LIN {X 0,Y 573.263,Z 117.071,A -85,B 0,C 180,E1 -2310.634,E2 -2310.634} C_VEL
LIN {X 0,Y 573.25,Z 117.074,A -85,B 0,C 180,E1 -2313.024,E2 -2313.024} C_VEL
LIN {X 0,Y 573.273,Z 117.075,A -85,B 0,C 180,E1 -2315.366,E2 -2315.366} C_VEL
LIN {X 0,Y 573.228,Z 117.075,A -85,B 0,C 180,E1 -2318.419,E2 -2318.419} C_VEL
LIN {X 0,Y 573.277,Z 117.069,A -85,B 0,C 180,E1 -2320.728,E2 -2320.728} C_VEL
LIN {X 0,Y 573.249,Z 117.079,A -85,B 0,C 180,E1 -2323.621,E2 -2323.621} C_VEL
LIN {X 0,Y 573.271,Z 117.074,A -85,B 0,C 180,E1 -2325.807,E2 -2325.807} C_VEL
LIN {X 0,Y 573.261,Z 117.073,A -85,B 0,C 180,E1 -2328.745,E2 -2328.745} C_VEL
LIN {X 0,Y 573.288,Z 117.073,A -85,B 0,C 180,E1 -2331.54,E2 -2331.54} C_VEL
LIN {X 0,Y 573.296,Z 117.068,A -85,B 0,C 180,E1 -2334.372,E2 -2334.372} C_VEL
LIN {X 0,Y 573.315,Z 117.066,A -85,B 0,C 180,E1 -2337.892,E2 -2337.892} C_VEL
LIN {X 0,Y 573.327,Z 117.067,A -85,B 0,C 180,E1 -2340.702,E2 -2340.702} C_VEL
LIN {X 0,Y 573.302,Z 117.073,A -85,B 0,C 180,E1 -2342.81,E2 -2342.81} C_VEL
LIN {X 0,Y 573.296,Z 117.068,A -85,B 0,C 180,E1 -2345.628,E2 -2345.628} C_VEL
LIN {X 0,Y 573.282,Z 117.073,A -85,B 0,C 180,E1 -2348.459,E2 -2348.459} C_VEL
LIN {X 0,Y 573.269,Z 117.073,A -85,B 0,C 180,E1 -2351.312,E2 -2351.312} C_VEL
LIN {X 0,Y 573.279,Z 117.074,A -85,B 0,C 180,E1 -2354.424,E2 -2354.424} C_VEL
LIN {X 0,Y 573.256,Z 117.076,A -85,B 0,C 180,E1 -2357.112,E2 -2357.112} C_VEL
LIN {X 0,Y 573.251,Z 117.075,A -85,B 0,C 180,E1 -2360.077,E2 -2360.077} C_VEL
LIN {X 0,Y 573.232,Z 117.078,A -85,B 0,C 180,E1 -2363.099,E2 -2363.099} C_VEL
LIN {X 0,Y 573.247,Z 117.079,A -85,B 0,C 180,E1 -2364.384,E2 -2364.384} C_VEL
LIN {X 0,Y 572.62,Z 117.161,A -85,B 0,C 180,E1 -2364.971,E2 -2364.971} C_VEL
LIN {X 0,Y 569.779,Z 117.514,A -85,B 0,C 180,E1 -2365.922,E2 -2365.922} C_VEL
LIN {X 0,Y 567.35,Z 117.815,A -85,B 0,C 180,E1 -2366.688,E2 -2366.688} C_VEL
LIN {X 0,Y 566.299,Z 117.941,A -85,B 0,C 180,E1 -2367.279,E2 -2367.279} C_VEL
LIN {X 0,Y 566.211,Z 117.951,A -85,B 0,C 180,E1 -2367.479,E2 -2367.479} C_VEL
LIN {X 0,Y 566.2,Z 117.954,A -85,B 0,C 180,E1 -2369.769,E2 -2369.769} C_VEL
LIN {X 0,Y 566.207,Z 117.96,A -85,B 0,C 180,E1 -2372.431,E2 -2372.431} C_VEL
LIN {X 0,Y 566.25,Z 118.059,A -85,B 0,C 180,E1 -2375.403,E2 -2375.403} C_VEL
LIN {X 0,Y 566.277,Z 127.449,A -85,B 0,C 180,E1 -2377.2,E2 -2377.2} C_VEL
LIN {X 0,Y 566.206,Z 137.001,A -85,B 0,C 180,E1 -2379.061,E2 -2379.061} C_VEL
LIN {X 0,Y 567.133,Z 143.743,A -85,B 0,C 180,E1 -2379.171,E2 -2379.171} C_VEL
LIN {X 0,Y 566.929,Z 243.631,A -85,B 0,C 180,E1 -2380.461,E2 -2380.461} C_VEL
LIN {X 0,Y 566.817,Z 257.421,A -85,B 0,C 180,E1 -2380.799,E2 -2380.799} C_VEL
LIN {X 0,Y 566.695,Z 270.238,A -85,B 0,C 180,E1 -2381.27,E2 -2381.27} C_VEL
LIN {X 0,Y 566.563,Z 282.807,A -85,B 0,C 180,E1 -2381.903,E2 -2381.903} C_VEL
LIN {X 0,Y 566.432,Z 294.236,A -85,B 0,C 180,E1 -2382.643,E2 -2382.643} C_VEL
LIN {X 0,Y 566.313,Z 303.744,A -85,B 0,C 180,E1 -2383.409,E2 -2383.409} C_VEL
LIN {X 0,Y 566.2,Z 312.297,A -85,B 0,C 180,E1 -2384.245,E2 -2384.245} C_VEL
LIN {X 0,Y 566.074,Z 320.91,A -85,B 0,C 180,E1 -2385.272,E2 -2385.272} C_VEL
LIN {X 0,Y 565.998,Z 327.798,A -85,B 0,C 180,E1 -2386.28,E2 -2386.28} C_VEL
LIN {X 0,Y 565.943,Z 334.451,A -85,B 0,C 180,E1 -2387.499,E2 -2387.499} C_VEL
LIN {X 0,Y 565.904,Z 339.904,A -85,B 0,C 180,E1 -2388.837,E2 -2388.837} C_VEL
LIN {X 0,Y 565.884,Z 342.757,A -85,B 0,C 180,E1 -2389.774,E2 -2389.774} C_VEL
LIN {X 0,Y 565.822,Z 344.826,A -85,B 0,C 180,E1 -2390.694,E2 -2390.694} C_VEL
LIN {X 0,Y 565.833,Z 346.17,A -85,B 0,C 180,E1 -2391.609,E2 -2391.609} C_VEL
LIN {X 0,Y 565.833,Z 346.918,A -85,B 0,C 180,E1 -2392.648,E2 -2392.648} C_VEL
LIN {X 0,Y 565.819,Z 346.731,A -85,B 0,C 180,E1 -2393.839,E2 -2393.839} C_VEL
LIN {X 0,Y 565.854,Z 345.231,A -85,B 0,C 180,E1 -2395.157,E2 -2395.157} C_VEL
LIN {X 0,Y 565.912,Z 342.766,A -85,B 0,C 180,E1 -2396.311,E2 -2396.311} C_VEL
LIN {X 0,Y 565.884,Z 338.589,A -85,B 0,C 180,E1 -2397.621,E2 -2397.621} C_VEL
LIN {X 0,Y 565.949,Z 334.579,A -85,B 0,C 180,E1 -2398.563,E2 -2398.563} C_VEL
LIN {X 0,Y 566.027,Z 329.057,A -85,B 0,C 180,E1 -2399.605,E2 -2399.605} C_VEL
LIN {X 0,Y 566.052,Z 322.317,A -85,B 0,C 180,E1 -2400.632,E2 -2400.632} C_VEL
LIN {X 0,Y 566.169,Z 313.849,A -85,B 0,C 180,E1 -2401.674,E2 -2401.674} C_VEL
LIN {X 0,Y 566.274,Z 303.927,A -85,B 0,C 180,E1 -2402.664,E2 -2402.664} C_VEL
LIN {X 0,Y 566.424,Z 293.916,A -85,B 0,C 180,E1 -2403.47,E2 -2403.47} C_VEL
LIN {X 0,Y 566.523,Z 283.148,A -85,B 0,C 180,E1 -2404.168,E2 -2404.168} C_VEL
LIN {X 0,Y 566.673,Z 271.108,A -85,B 0,C 180,E1 -2404.781,E2 -2404.781} C_VEL
LIN {X 0,Y 566.809,Z 259.887,A -85,B 0,C 180,E1 -2405.213,E2 -2405.213} C_VEL
LIN {X 0,Y 566.924,Z 247.085,A -85,B 0,C 180,E1 -2405.56,E2 -2405.56} C_VEL
LIN {X 0,Y 566.991,Z 231.232,A -85,B 0,C 180,E1 -2405.807,E2 -2405.807} C_VEL
LIN {X 0,Y 567.066,Z 141.922,A -85,B 0,C 180,E1 -2406.944,E2 -2406.944} C_VEL
LIN {X 0,Y 566.199,Z 136.958,A -85,B 0,C 180,E1 -2407.032,E2 -2407.032} C_VEL
LIN {X 0,Y 566.329,Z 121.586,A -85,B 0,C 180,E1 -2410.046,E2 -2410.046} C_VEL
LIN {X 0,Y 566.237,Z 117.951,A -85,B 0,C 180,E1 -2410.789,E2 -2410.789} C_VEL
LIN {X 0,Y 566.209,Z 117.956,A -85,B 0,C 180,E1 -2413.412,E2 -2413.412} C_VEL
LIN {X 0,Y 566.192,Z 117.954,A -85,B 0,C 180,E1 -2416.359,E2 -2416.359} C_VEL
LIN {X 0,Y 566.235,Z 117.947,A -85,B 0,C 180,E1 -2418.675,E2 -2418.675} C_VEL
LIN {X 0,Y 566.226,Z 117.956,A -85,B 0,C 180,E1 -2421.434,E2 -2421.434} C_VEL
LIN {X 0,Y 566.259,Z 117.944,A -85,B 0,C 180,E1 -2424.302,E2 -2424.302} C_VEL
LIN {X 0,Y 566.287,Z 117.943,A -85,B 0,C 180,E1 -2427.866,E2 -2427.866} C_VEL
LIN {X 0,Y 566.294,Z 117.941,A -85,B 0,C 180,E1 -2430.711,E2 -2430.711} C_VEL
LIN {X 0,Y 566.265,Z 117.946,A -85,B 0,C 180,E1 -2432.846,E2 -2432.846} C_VEL
LIN {X 0,Y 566.265,Z 117.946,A -85,B 0,C 180,E1 -2435.698,E2 -2435.698} C_VEL
LIN {X 0,Y 566.205,Z 117.952,A -85,B 0,C 180,E1 -2438.566,E2 -2438.566} C_VEL
LIN {X 0,Y 566.243,Z 117.95,A -85,B 0,C 180,E1 -2441.454,E2 -2441.454} C_VEL
LIN {X 0,Y 566.235,Z 117.95,A -85,B 0,C 180,E1 -2444.506,E2 -2444.506} C_VEL
LIN {X 0,Y 566.197,Z 117.955,A -85,B 0,C 180,E1 -2447.332,E2 -2447.332} C_VEL
LIN {X 0,Y 566.206,Z 117.953,A -85,B 0,C 180,E1 -2450.337,E2 -2450.337} C_VEL
LIN {X 0,Y 566.171,Z 117.957,A -85,B 0,C 180,E1 -2453.281,E2 -2453.281} C_VEL
LIN {X 0,Y 566.209,Z 117.95,A -85,B 0,C 180,E1 -2455.749,E2 -2455.749} C_VEL
LIN {X 0,Y 566.202,Z 117.954,A -85,B 0,C 180,E1 -2458.202,E2 -2458.202} C_VEL
LIN {X 0,Y 566.189,Z 117.955,A -85,B 0,C 180,E1 -2461.076,E2 -2461.076} C_VEL
LIN {X 0,Y 566.196,Z 117.952,A -85,B 0,C 180,E1 -2463.732,E2 -2463.732} C_VEL
LIN {X 0,Y 566.199,Z 117.959,A -85,B 0,C 180,E1 -2466.57,E2 -2466.57} C_VEL
LIN {X 0,Y 566.214,Z 117.95,A -85,B 0,C 180,E1 -2469.686,E2 -2469.686} C_VEL
LIN {X 0,Y 566.21,Z 117.956,A -85,B 0,C 180,E1 -2472.087,E2 -2472.087} C_VEL
LIN {X 0,Y 566.172,Z 117.955,A -85,B 0,C 180,E1 -2475.036,E2 -2475.036} C_VEL
LIN {X 0,Y 566.188,Z 117.959,A -85,B 0,C 180,E1 -2477.91,E2 -2477.91} C_VEL
LIN {X 0,Y 566.221,Z 117.95,A -85,B 0,C 180,E1 -2480.727,E2 -2480.727} C_VEL
LIN {X 0,Y 566.2,Z 117.957,A -85,B 0,C 180,E1 -2483.786,E2 -2483.786} C_VEL
LIN {X 0,Y 566.209,Z 117.955,A -85,B 0,C 180,E1 -2486.266,E2 -2486.266} C_VEL
LIN {X 0,Y 566.196,Z 117.952,A -85,B 0,C 180,E1 -2488.922,E2 -2488.922} C_VEL
LIN {X 0,Y 566.191,Z 117.953,A -85,B 0,C 180,E1 -2491.047,E2 -2491.047} C_VEL
LIN {X 0,Y 566.214,Z 117.954,A -85,B 0,C 180,E1 -2493.459,E2 -2493.459} C_VEL
LIN {X 0,Y 566.195,Z 117.96,A -85,B 0,C 180,E1 -2495.819,E2 -2495.819} C_VEL
LIN {X 0,Y 566.207,Z 117.951,A -85,B 0,C 180,E1 -2498.902,E2 -2498.902} C_VEL
LIN {X 0,Y 566.205,Z 117.954,A -85,B 0,C 180,E1 -2501.172,E2 -2501.172} C_VEL
LIN {X 0,Y 566.214,Z 117.958,A -85,B 0,C 180,E1 -2503.412,E2 -2503.412} C_VEL
LIN {X 0,Y 566.195,Z 117.952,A -85,B 0,C 180,E1 -2506.359,E2 -2506.359} C_VEL
LIN {X 0,Y 566.233,Z 117.948,A -85,B 0,C 180,E1 -2508.675,E2 -2508.675} C_VEL
LIN {X 0,Y 566.232,Z 117.955,A -85,B 0,C 180,E1 -2511.435,E2 -2511.435} C_VEL
LIN {X 0,Y 566.264,Z 117.943,A -85,B 0,C 180,E1 -2514.302,E2 -2514.302} C_VEL
LIN {X 0,Y 566.285,Z 117.941,A -85,B 0,C 180,E1 -2517.866,E2 -2517.866} C_VEL
LIN {X 0,Y 566.298,Z 117.943,A -85,B 0,C 180,E1 -2520.711,E2 -2520.711} C_VEL
LIN {X 0,Y 566.269,Z 117.949,A -85,B 0,C 180,E1 -2522.846,E2 -2522.846} C_VEL
LIN {X 0,Y 566.265,Z 117.944,A -85,B 0,C 180,E1 -2525.698,E2 -2525.698} C_VEL
LIN {X 0,Y 566.226,Z 117.953,A -85,B 0,C 180,E1 -2528.566,E2 -2528.566} C_VEL
LIN {X 0,Y 566.241,Z 117.947,A -85,B 0,C 180,E1 -2531.455,E2 -2531.455} C_VEL
LIN {X 0,Y 566.233,Z 117.953,A -85,B 0,C 180,E1 -2534.507,E2 -2534.507} C_VEL
LIN {X 0,Y 566.198,Z 117.952,A -85,B 0,C 180,E1 -2537.332,E2 -2537.332} C_VEL
LIN {X 0,Y 566.213,Z 117.955,A -85,B 0,C 180,E1 -2540.337,E2 -2540.337} C_VEL
LIN {X 0,Y 566.172,Z 117.955,A -85,B 0,C 180,E1 -2543.282,E2 -2543.282} C_VEL
LIN {X 0,Y 566.214,Z 117.95,A -85,B 0,C 180,E1 -2545.749,E2 -2545.749} C_VEL
LIN {X 0,Y 566.202,Z 117.957,A -85,B 0,C 180,E1 -2548.202,E2 -2548.202} C_VEL
LIN {X 0,Y 566.194,Z 117.952,A -85,B 0,C 180,E1 -2551.077,E2 -2551.077} C_VEL
LIN {X 0,Y 566.211,Z 117.952,A -85,B 0,C 180,E1 -2553.734,E2 -2553.734} C_VEL
LIN {X 0,Y 566.2,Z 117.955,A -85,B 0,C 180,E1 -2556.57,E2 -2556.57} C_VEL
LIN {X 0,Y 566.222,Z 117.949,A -85,B 0,C 180,E1 -2559.273,E2 -2559.273} C_VEL
LIN {X 0,Y 566.214,Z 117.959,A -85,B 0,C 180,E1 -2562.088,E2 -2562.088} C_VEL
LIN {X 0,Y 566.174,Z 117.954,A -85,B 0,C 180,E1 -2565.036,E2 -2565.036} C_VEL
LIN {X 0,Y 566.219,Z 117.955,A -85,B 0,C 180,E1 -2568.136,E2 -2568.136} C_VEL
LIN {X 0,Y 566.223,Z 117.948,A -85,B 0,C 180,E1 -2570.727,E2 -2570.727} C_VEL
LIN {X 0,Y 566.185,Z 117.963,A -85,B 0,C 180,E1 -2573.789,E2 -2573.789} C_VEL
LIN {X 0,Y 566.213,Z 117.951,A -85,B 0,C 180,E1 -2576.266,E2 -2576.266} C_VEL
LIN {X 0,Y 566.192,Z 117.953,A -85,B 0,C 180,E1 -2578.924,E2 -2578.924} C_VEL
LIN {X 0,Y 566.214,Z 117.956,A -85,B 0,C 180,E1 -2581.858,E2 -2581.858} C_VEL
LIN {X 0,Y 566.215,Z 117.953,A -85,B 0,C 180,E1 -2584.251,E2 -2584.251} C_VEL
LIN {X 0,Y 566.276,Z 118.069,A -85,B 0,C 180,E1 -2585.628,E2 -2585.628} C_VEL
LIN {X 0,Y 567.118,Z 124.11,A -85,B 0,C 180,E1 -2586.498,E2 -2586.498} C_VEL
LIN {X 0,Y 566.895,Z 141.853,A -85,B 0,C 180,E1 -2588.929,E2 -2588.929} C_VEL
LIN {X 0,Y 566.77,Z 162.723,A -85,B 0,C 180,E1 -2591.754,E2 -2591.754} C_VEL
LIN {X 0,Y 566.5,Z 183.519,A -85,B 0,C 180,E1 -2594.53,E2 -2594.53} C_VEL
LIN {X 0,Y 566.428,Z 194.355,A -85,B 0,C 180,E1 -2595.987,E2 -2595.987} C_VEL
LIN {X 0,Y 567.152,Z 200.513,A -85,B 0,C 180,E1 -2596.085,E2 -2596.085} C_VEL
LIN {X 0,Y 566.964,Z 302.949,A -85,B 0,C 180,E1 -2597.403,E2 -2597.403} C_VEL
LIN {X 0,Y 566.839,Z 316.219,A -85,B 0,C 180,E1 -2597.719,E2 -2597.719} C_VEL
LIN {X 0,Y 566.764,Z 328.379,A -85,B 0,C 180,E1 -2598.149,E2 -2598.149} C_VEL
LIN {X 0,Y 566.603,Z 340.24,A -85,B 0,C 180,E1 -2598.713,E2 -2598.713} C_VEL
LIN {X 0,Y 566.439,Z 352.196,A -85,B 0,C 180,E1 -2599.455,E2 -2599.455} C_VEL
LIN {X 0,Y 566.325,Z 362.605,A -85,B 0,C 180,E1 -2600.265,E2 -2600.265} C_VEL
LIN {X 0,Y 566.207,Z 371.113,A -85,B 0,C 180,E1 -2601.074,E2 -2601.074} C_VEL
LIN {X 0,Y 566.112,Z 378.961,A -85,B 0,C 180,E1 -2601.972,E2 -2601.972} C_VEL
LIN {X 0,Y 566.004,Z 386.623,A -85,B 0,C 180,E1 -2603.047,E2 -2603.047} C_VEL
LIN {X 0,Y 566.004,Z 393.68,A -85,B 0,C 180,E1 -2604.299,E2 -2604.299} C_VEL
LIN {X 0,Y 565.933,Z 398.373,A -85,B 0,C 180,E1 -2605.37,E2 -2605.37} C_VEL
LIN {X 0,Y 565.927,Z 401.958,A -85,B 0,C 180,E1 -2606.44,E2 -2606.44} C_VEL
LIN {X 0,Y 565.878,Z 403.807,A -85,B 0,C 180,E1 -2607.152,E2 -2607.152} C_VEL
LIN {X 0,Y 565.846,Z 406.184,A -85,B 0,C 180,E1 -2608.577,E2 -2608.577} C_VEL
LIN {X 0,Y 565.839,Z 407,A -85,B 0,C 180,E1 -2610,E2 -2610} C_VEL
LIN {X 0,Y 565.846,Z 406.185,A -85,B 0,C 180,E1 -2611.423,E2 -2611.423} C_VEL
LIN {X 0,Y 565.878,Z 403.81,A -85,B 0,C 180,E1 -2612.847,E2 -2612.847} C_VEL
LIN {X 0,Y 565.926,Z 400.896,A -85,B 0,C 180,E1 -2613.916,E2 -2613.916} C_VEL
LIN {X 0,Y 565.878,Z 396.949,A -85,B 0,C 180,E1 -2614.987,E2 -2614.987} C_VEL
LIN {X 0,Y 566.002,Z 391.867,A -85,B 0,C 180,E1 -2616.058,E2 -2616.058} C_VEL
LIN {X 0,Y 566.04,Z 385.468,A -85,B 0,C 180,E1 -2617.132,E2 -2617.132} C_VEL
LIN {X 0,Y 566.134,Z 377.478,A -85,B 0,C 180,E1 -2618.208,E2 -2618.208} C_VEL
LIN {X 0,Y 566.229,Z 369.335,A -85,B 0,C 180,E1 -2619.105,E2 -2619.105} C_VEL
LIN {X 0,Y 566.347,Z 359.4,A -85,B 0,C 180,E1 -2620.005,E2 -2620.005} C_VEL
LIN {X 0,Y 566.536,Z 348.292,A -85,B 0,C 180,E1 -2620.807,E2 -2620.807} C_VEL
LIN {X 0,Y 566.613,Z 337.175,A -85,B 0,C 180,E1 -2621.447,E2 -2621.447} C_VEL
LIN {X 0,Y 566.776,Z 324.981,A -85,B 0,C 180,E1 -2621.987,E2 -2621.987} C_VEL
LIN {X 0,Y 566.917,Z 312.178,A -85,B 0,C 180,E1 -2622.393,E2 -2622.393} C_VEL
LIN {X 0,Y 566.993,Z 300.111,A -85,B 0,C 180,E1 -2622.642,E2 -2622.642} C_VEL
LIN {X 0,Y 567.038,Z 198.729,A -85,B 0,C 180,E1 -2623.94,E2 -2623.94} C_VEL
LIN {X 0,Y 566.428,Z 194.27,A -85,B 0,C 180,E1 -2624.024,E2 -2624.024} C_VEL
LIN {X 0,Y 566.62,Z 172.717,A -85,B 0,C 180,E1 -2626.902,E2 -2626.902} C_VEL
LIN {X 0,Y 566.763,Z 152.969,A -85,B 0,C 180,E1 -2629.538,E2 -2629.538} C_VEL
LIN {X 0,Y 566.976,Z 133.142,A -85,B 0,C 180,E1 -2632.214,E2 -2632.214} C_VEL
LIN {X 0,Y 566.964,Z 121.783,A -85,B 0,C 180,E1 -2633.765,E2 -2633.765} C_VEL
LIN {X 0,Y 566.263,Z 117.955,A -85,B 0,C 180,E1 -2634.324,E2 -2634.324} C_VEL
LIN {X 0,Y 566.213,Z 117.951,A -85,B 0,C 180,E1 -2637.339,E2 -2637.339} C_VEL
LIN {X 0,Y 566.203,Z 117.954,A -85,B 0,C 180,E1 -2639.768,E2 -2639.768} C_VEL
LIN {X 0,Y 566.207,Z 117.96,A -85,B 0,C 180,E1 -2642.43,E2 -2642.43} C_VEL
LIN {X 0,Y 566.181,Z 117.955,A -85,B 0,C 180,E1 -2644.989,E2 -2644.989} C_VEL
LIN {X 0,Y 566.198,Z 117.953,A -85,B 0,C 180,E1 -2647.46,E2 -2647.46} C_VEL
LIN {X 0,Y 566.228,Z 117.958,A -85,B 0,C 180,E1 -2650.197,E2 -2650.197} C_VEL
LIN {X 0,Y 566.202,Z 117.952,A -85,B 0,C 180,E1 -2653.054,E2 -2653.054} C_VEL
LIN {X 0,Y 566.199,Z 117.961,A -85,B 0,C 180,E1 -2656.048,E2 -2656.048} C_VEL
LIN {X 0,Y 566.212,Z 117.95,A -85,B 0,C 180,E1 -2658.863,E2 -2658.863} C_VEL
LIN {X 0,Y 566.19,Z 117.957,A -85,B 0,C 180,E1 -2661.637,E2 -2661.637} C_VEL
LIN {X 0,Y 566.161,Z 117.959,A -85,B 0,C 180,E1 -2664.308,E2 -2664.308} C_VEL
LIN {X 0,Y 566.22,Z 117.948,A -85,B 0,C 180,E1 -2666.898,E2 -2666.898} C_VEL
LIN {X 0,Y 566.183,Z 117.958,A -85,B 0,C 180,E1 -2669.407,E2 -2669.407} C_VEL
LIN {X 0,Y 566.21,Z 117.957,A -85,B 0,C 180,E1 -2671.857,E2 -2671.857} C_VEL
LIN {X 0,Y 566.213,Z 117.95,A -85,B 0,C 180,E1 -2674.251,E2 -2674.251} C_VEL
LIN {X 0,Y 566.168,Z 117.955,A -85,B 0,C 180,E1 -2676.719,E2 -2676.719} C_VEL
LIN {X 0,Y 566.213,Z 117.956,A -85,B 0,C 180,E1 -2679.663,E2 -2679.663} C_VEL
LIN {X 0,Y 566.198,Z 117.952,A -85,B 0,C 180,E1 -2682.668,E2 -2682.668} C_VEL
LIN {X 0,Y 566.232,Z 117.953,A -85,B 0,C 180,E1 -2685.627,E2 -2685.627} C_VEL
LIN {X 0,Y 566.233,Z 117.948,A -85,B 0,C 180,E1 -2688.675,E2 -2688.675} C_VEL
LIN {X 0,Y 566.232,Z 117.953,A -85,B 0,C 180,E1 -2691.434,E2 -2691.434} C_VEL
LIN {X 0,Y 566.265,Z 117.943,A -85,B 0,C 180,E1 -2694.302,E2 -2694.302} C_VEL
LIN {X 0,Y 566.285,Z 117.941,A -85,B 0,C 180,E1 -2697.866,E2 -2697.866} C_VEL
LIN {X 0,Y 566.298,Z 117.943,A -85,B 0,C 180,E1 -2700.711,E2 -2700.711} C_VEL
LIN {X 0,Y 566.269,Z 117.95,A -85,B 0,C 180,E1 -2702.845,E2 -2702.845} C_VEL
LIN {X 0,Y 566.264,Z 117.943,A -85,B 0,C 180,E1 -2705.698,E2 -2705.698} C_VEL
LIN {X 0,Y 566.226,Z 117.953,A -85,B 0,C 180,E1 -2708.566,E2 -2708.566} C_VEL
LIN {X 0,Y 566.24,Z 117.947,A -85,B 0,C 180,E1 -2711.454,E2 -2711.454} C_VEL
LIN {X 0,Y 566.232,Z 117.954,A -85,B 0,C 180,E1 -2714.507,E2 -2714.507} C_VEL
LIN {X 0,Y 566.197,Z 117.953,A -85,B 0,C 180,E1 -2717.332,E2 -2717.332} C_VEL
LIN {X 0,Y 566.212,Z 117.956,A -85,B 0,C 180,E1 -2720.337,E2 -2720.337} C_VEL
LIN {X 0,Y 566.17,Z 117.957,A -85,B 0,C 180,E1 -2723.282,E2 -2723.282} C_VEL
LIN {X 0,Y 566.212,Z 117.952,A -85,B 0,C 180,E1 -2725.749,E2 -2725.749} C_VEL
LIN {X 0,Y 566.211,Z 117.951,A -85,B 0,C 180,E1 -2727.479,E2 -2727.479} C_VEL
LIN {X 0,Y 565.534,Z 118.041,A -85,B 0,C 180,E1 -2728.073,E2 -2728.073} C_VEL
LIN {X 0,Y 562.665,Z 118.397,A -85,B 0,C 180,E1 -2729.036,E2 -2729.036} C_VEL
LIN {X 0,Y 560.251,Z 118.698,A -85,B 0,C 180,E1 -2729.812,E2 -2729.812} C_VEL
LIN {X 0,Y 559.222,Z 118.83,A -85,B 0,C 180,E1 -2730.41,E2 -2730.41} C_VEL
LIN {X 0,Y 559.143,Z 118.834,A -85,B 0,C 180,E1 -2730.613,E2 -2730.613} C_VEL
LIN {X 0,Y 559.174,Z 118.832,A -85,B 0,C 180,E1 -2732.714,E2 -2732.714} C_VEL
LIN {X 0,Y 559.233,Z 118.95,A -85,B 0,C 180,E1 -2735.344,E2 -2735.344} C_VEL
LIN {X 0,Y 559.315,Z 126.341,A -85,B 0,C 180,E1 -2736.753,E2 -2736.753} C_VEL
LIN {X 0,Y 559.239,Z 137.251,A -85,B 0,C 180,E1 -2738.873,E2 -2738.873} C_VEL
LIN {X 0,Y 560.266,Z 144.433,A -85,B 0,C 180,E1 -2739.003,E2 -2739.003} C_VEL
LIN {X 0,Y 560.015,Z 243.987,A -85,B 0,C 180,E1 -2740.307,E2 -2740.307} C_VEL
LIN {X 0,Y 559.873,Z 257.853,A -85,B 0,C 180,E1 -2740.653,E2 -2740.653} C_VEL
LIN {X 0,Y 559.762,Z 270.366,A -85,B 0,C 180,E1 -2741.122,E2 -2741.122} C_VEL
LIN {X 0,Y 559.585,Z 282.373,A -85,B 0,C 180,E1 -2741.732,E2 -2741.732} C_VEL
LIN {X 0,Y 559.429,Z 294.022,A -85,B 0,C 180,E1 -2742.493,E2 -2742.493} C_VEL
LIN {X 0,Y 559.289,Z 303.86,A -85,B 0,C 180,E1 -2743.298,E2 -2743.298} C_VEL
LIN {X 0,Y 559.139,Z 313.237,A -85,B 0,C 180,E1 -2744.238,E2 -2744.238} C_VEL
LIN {X 0,Y 559.023,Z 321.476,A -85,B 0,C 180,E1 -2745.249,E2 -2745.249} C_VEL
LIN {X 0,Y 558.929,Z 328.114,A -85,B 0,C 180,E1 -2746.246,E2 -2746.246} C_VEL
LIN {X 0,Y 558.861,Z 333.466,A -85,B 0,C 180,E1 -2747.229,E2 -2747.229} C_VEL
LIN {X 0,Y 558.829,Z 337.755,A -85,B 0,C 180,E1 -2748.2,E2 -2748.2} C_VEL
LIN {X 0,Y 558.804,Z 341.126,A -85,B 0,C 180,E1 -2749.157,E2 -2749.157} C_VEL
LIN {X 0,Y 558.764,Z 343.682,A -85,B 0,C 180,E1 -2750.107,E2 -2750.107} C_VEL
LIN {X 0,Y 558.731,Z 345.764,A -85,B 0,C 180,E1 -2751.248,E2 -2751.248} C_VEL
LIN {X 0,Y 558.74,Z 346.844,A -85,B 0,C 180,E1 -2752.413,E2 -2752.413} C_VEL
LIN {X 0,Y 558.722,Z 346.791,A -85,B 0,C 180,E1 -2753.758,E2 -2753.758} C_VEL
LIN {X 0,Y 558.754,Z 345.762,A -85,B 0,C 180,E1 -2754.842,E2 -2754.842} C_VEL
LIN {X 0,Y 558.803,Z 343.376,A -85,B 0,C 180,E1 -2756.106,E2 -2756.106} C_VEL
LIN {X 0,Y 558.796,Z 339.508,A -85,B 0,C 180,E1 -2757.422,E2 -2757.422} C_VEL
LIN {X 0,Y 558.853,Z 335.291,A -85,B 0,C 180,E1 -2758.474,E2 -2758.474} C_VEL
LIN {X 0,Y 558.942,Z 329.57,A -85,B 0,C 180,E1 -2759.596,E2 -2759.596} C_VEL
LIN {X 0,Y 558.974,Z 322.965,A -85,B 0,C 180,E1 -2760.637,E2 -2760.637} C_VEL
LIN {X 0,Y 559.127,Z 314.068,A -85,B 0,C 180,E1 -2761.759,E2 -2761.759} C_VEL
LIN {X 0,Y 559.244,Z 304.878,A -85,B 0,C 180,E1 -2762.697,E2 -2762.697} C_VEL
LIN {X 0,Y 559.413,Z 295.136,A -85,B 0,C 180,E1 -2763.513,E2 -2763.513} C_VEL
LIN {X 0,Y 559.523,Z 284.746,A -85,B 0,C 180,E1 -2764.221,E2 -2764.221} C_VEL
LIN {X 0,Y 559.703,Z 272.704,A -85,B 0,C 180,E1 -2764.861,E2 -2764.861} C_VEL
LIN {X 0,Y 559.857,Z 261.062,A -85,B 0,C 180,E1 -2765.33,E2 -2765.33} C_VEL
LIN {X 0,Y 560.004,Z 248.794,A -85,B 0,C 180,E1 -2765.683,E2 -2765.683} C_VEL
LIN {X 0,Y 560.114,Z 235.741,A -85,B 0,C 180,E1 -2765.909,E2 -2765.909} C_VEL
LIN {X 0,Y 560.177,Z 142.601,A -85,B 0,C 180,E1 -2767.112,E2 -2767.112} C_VEL
LIN {X 0,Y 559.179,Z 137.233,A -85,B 0,C 180,E1 -2767.216,E2 -2767.216} C_VEL
LIN {X 0,Y 559.325,Z 122.154,A -85,B 0,C 180,E1 -2770.168,E2 -2770.168} C_VEL
LIN {X 0,Y 559.211,Z 118.827,A -85,B 0,C 180,E1 -2770.838,E2 -2770.838} C_VEL
LIN {X 0,Y 559.16,Z 118.836,A -85,B 0,C 180,E1 -2773.948,E2 -2773.948} C_VEL
LIN {X 0,Y 559.168,Z 118.831,A -85,B 0,C 180,E1 -2776.184,E2 -2776.184} C_VEL
LIN {X 0,Y 559.195,Z 118.826,A -85,B 0,C 180,E1 -2779.134,E2 -2779.134} C_VEL
LIN {X 0,Y 559.199,Z 118.826,A -85,B 0,C 180,E1 -2782.054,E2 -2782.054} C_VEL
LIN {X 0,Y 559.253,Z 118.819,A -85,B 0,C 180,E1 -2784.953,E2 -2784.953} C_VEL
LIN {X 0,Y 559.257,Z 118.819,A -85,B 0,C 180,E1 -2787.839,E2 -2787.839} C_VEL
LIN {X 0,Y 559.266,Z 118.816,A -85,B 0,C 180,E1 -2790.72,E2 -2790.72} C_VEL
LIN {X 0,Y 559.232,Z 118.823,A -85,B 0,C 180,E1 -2792.881,E2 -2792.881} C_VEL
LIN {X 0,Y 559.233,Z 118.821,A -85,B 0,C 180,E1 -2795.77,E2 -2795.77} C_VEL
LIN {X 0,Y 559.17,Z 118.83,A -85,B 0,C 180,E1 -2798.675,E2 -2798.675} C_VEL
LIN {X 0,Y 559.206,Z 118.824,A -85,B 0,C 180,E1 -2801.6,E2 -2801.6} C_VEL
LIN {X 0,Y 559.201,Z 118.827,A -85,B 0,C 180,E1 -2804.595,E2 -2804.595} C_VEL
LIN {X 0,Y 559.14,Z 118.832,A -85,B 0,C 180,E1 -2807.557,E2 -2807.557} C_VEL
LIN {X 0,Y 559.165,Z 118.827,A -85,B 0,C 180,E1 -2809.838,E2 -2809.838} C_VEL
LIN {X 0,Y 559.141,Z 118.832,A -85,B 0,C 180,E1 -2812.153,E2 -2812.153} C_VEL
LIN {X 0,Y 559.175,Z 118.828,A -85,B 0,C 180,E1 -2815.298,E2 -2815.298} C_VEL
LIN {X 0,Y 559.156,Z 118.829,A -85,B 0,C 180,E1 -2817.713,E2 -2817.713} C_VEL
LIN {X 0,Y 559.15,Z 118.833,A -85,B 0,C 180,E1 -2820.183,E2 -2820.183} C_VEL
LIN {X 0,Y 559.152,Z 118.836,A -85,B 0,C 180,E1 -2822.715,E2 -2822.715} C_VEL
LIN {X 0,Y 559.126,Z 118.833,A -85,B 0,C 180,E1 -2825.324,E2 -2825.324} C_VEL
LIN {X 0,Y 559.132,Z 118.835,A -85,B 0,C 180,E1 -2828.017,E2 -2828.017} C_VEL
LIN {X 0,Y 559.156,Z 118.831,A -85,B 0,C 180,E1 -2830.812,E2 -2830.812} C_VEL
LIN {X 0,Y 559.146,Z 118.83,A -85,B 0,C 180,E1 -2833.197,E2 -2833.197} C_VEL
LIN {X 0,Y 559.158,Z 118.837,A -85,B 0,C 180,E1 -2836.268,E2 -2836.268} C_VEL
LIN {X 0,Y 559.172,Z 118.827,A -85,B 0,C 180,E1 -2839.189,E2 -2839.189} C_VEL
LIN {X 0,Y 559.133,Z 118.84,A -85,B 0,C 180,E1 -2841.983,E2 -2841.983} C_VEL
LIN {X 0,Y 559.143,Z 118.831,A -85,B 0,C 180,E1 -2844.785,E2 -2844.785} C_VEL
LIN {X 0,Y 559.154,Z 118.831,A -85,B 0,C 180,E1 -2847.364,E2 -2847.364} C_VEL
LIN {X 0,Y 559.187,Z 118.83,A -85,B 0,C 180,E1 -2850.135,E2 -2850.135} C_VEL
LIN {X 0,Y 559.169,Z 118.829,A -85,B 0,C 180,E1 -2853.172,E2 -2853.172} C_VEL
LIN {X 0,Y 559.154,Z 118.835,A -85,B 0,C 180,E1 -2855.495,E2 -2855.495} C_VEL
LIN {X 0,Y 559.17,Z 118.827,A -85,B 0,C 180,E1 -2858.624,E2 -2858.624} C_VEL
LIN {X 0,Y 559.167,Z 118.828,A -85,B 0,C 180,E1 -2860.926,E2 -2860.926} C_VEL
LIN {X 0,Y 559.165,Z 118.831,A -85,B 0,C 180,E1 -2863.948,E2 -2863.948} C_VEL
LIN {X 0,Y 559.17,Z 118.828,A -85,B 0,C 180,E1 -2866.184,E2 -2866.184} C_VEL
LIN {X 0,Y 559.195,Z 118.83,A -85,B 0,C 180,E1 -2869.134,E2 -2869.134} C_VEL
LIN {X 0,Y 559.204,Z 118.823,A -85,B 0,C 180,E1 -2872.054,E2 -2872.054} C_VEL
LIN {X 0,Y 559.254,Z 118.822,A -85,B 0,C 180,E1 -2874.953,E2 -2874.953} C_VEL
LIN {X 0,Y 559.255,Z 118.817,A -85,B 0,C 180,E1 -2877.84,E2 -2877.84} C_VEL
LIN {X 0,Y 559.269,Z 118.819,A -85,B 0,C 180,E1 -2880.72,E2 -2880.72} C_VEL
LIN {X 0,Y 559.236,Z 118.826,A -85,B 0,C 180,E1 -2882.882,E2 -2882.882} C_VEL
LIN {X 0,Y 559.233,Z 118.819,A -85,B 0,C 180,E1 -2885.77,E2 -2885.77} C_VEL
LIN {X 0,Y 559.185,Z 118.831,A -85,B 0,C 180,E1 -2888.675,E2 -2888.675} C_VEL
LIN {X 0,Y 559.204,Z 118.823,A -85,B 0,C 180,E1 -2891.601,E2 -2891.601} C_VEL
LIN {X 0,Y 559.199,Z 118.831,A -85,B 0,C 180,E1 -2894.596,E2 -2894.596} C_VEL
LIN {X 0,Y 559.158,Z 118.828,A -85,B 0,C 180,E1 -2897.557,E2 -2897.557} C_VEL
LIN {X 0,Y 559.171,Z 118.827,A -85,B 0,C 180,E1 -2899.838,E2 -2899.838} C_VEL
LIN {X 0,Y 559.141,Z 118.834,A -85,B 0,C 180,E1 -2902.153,E2 -2902.153} C_VEL
LIN {X 0,Y 559.175,Z 118.826,A -85,B 0,C 180,E1 -2905.298,E2 -2905.298} C_VEL
LIN {X 0,Y 559.157,Z 118.829,A -85,B 0,C 180,E1 -2907.714,E2 -2907.714} C_VEL
LIN {X 0,Y 559.154,Z 118.836,A -85,B 0,C 180,E1 -2910.183,E2 -2910.183} C_VEL
LIN {X 0,Y 559.157,Z 118.832,A -85,B 0,C 180,E1 -2912.715,E2 -2912.715} C_VEL
LIN {X 0,Y 559.127,Z 118.832,A -85,B 0,C 180,E1 -2915.324,E2 -2915.324} C_VEL
LIN {X 0,Y 559.136,Z 118.839,A -85,B 0,C 180,E1 -2918.018,E2 -2918.018} C_VEL
LIN {X 0,Y 559.177,Z 118.827,A -85,B 0,C 180,E1 -2920.811,E2 -2920.811} C_VEL
LIN {X 0,Y 559.142,Z 118.836,A -85,B 0,C 180,E1 -2923.734,E2 -2923.734} C_VEL
LIN {X 0,Y 559.147,Z 118.83,A -85,B 0,C 180,E1 -2926.804,E2 -2926.804} C_VEL
LIN {X 0,Y 559.178,Z 118.827,A -85,B 0,C 180,E1 -2929.19,E2 -2929.19} C_VEL
LIN {X 0,Y 559.137,Z 118.838,A -85,B 0,C 180,E1 -2931.983,E2 -2931.983} C_VEL
LIN {X 0,Y 559.133,Z 118.832,A -85,B 0,C 180,E1 -2934.787,E2 -2934.787} C_VEL
LIN {X 0,Y 559.158,Z 118.833,A -85,B 0,C 180,E1 -2937.365,E2 -2937.365} C_VEL
LIN {X 0,Y 559.15,Z 118.833,A -85,B 0,C 180,E1 -2940.143,E2 -2940.143} C_VEL
LIN {X 0,Y 559.172,Z 118.832,A -85,B 0,C 180,E1 -2943.098,E2 -2943.098} C_VEL
LIN {X 0,Y 559.234,Z 118.946,A -85,B 0,C 180,E1 -2945.474,E2 -2945.474} C_VEL
LIN {X 0,Y 560.173,Z 124.747,A -85,B 0,C 180,E1 -2946.33,E2 -2946.33} C_VEL
LIN {X 0,Y 559.947,Z 141.506,A -85,B 0,C 180,E1 -2948.655,E2 -2948.655} C_VEL
LIN {X 0,Y 559.762,Z 161.003,A -85,B 0,C 180,E1 -2951.327,E2 -2951.327} C_VEL
LIN {X 0,Y 559.533,Z 180.436,A -85,B 0,C 180,E1 -2953.959,E2 -2953.959} C_VEL
LIN {X 0,Y 559.413,Z 194.196,A -85,B 0,C 180,E1 -2955.808,E2 -2955.808} C_VEL
LIN {X 0,Y 560.265,Z 202.109,A -85,B 0,C 180,E1 -2955.934,E2 -2955.934} C_VEL
LIN {X 0,Y 560.037,Z 302.947,A -85,B 0,C 180,E1 -2957.245,E2 -2957.245} C_VEL
LIN {X 0,Y 559.899,Z 316.218,A -85,B 0,C 180,E1 -2957.564,E2 -2957.564} C_VEL
LIN {X 0,Y 559.81,Z 328.377,A -85,B 0,C 180,E1 -2957.999,E2 -2957.999} C_VEL
LIN {X 0,Y 559.643,Z 340.057,A -85,B 0,C 180,E1 -2958.56,E2 -2958.56} C_VEL
LIN {X 0,Y 559.458,Z 352.194,A -85,B 0,C 180,E1 -2959.322,E2 -2959.322} C_VEL
LIN {X 0,Y 559.305,Z 362.606,A -85,B 0,C 180,E1 -2960.142,E2 -2960.142} C_VEL
LIN {X 0,Y 559.162,Z 371.114,A -85,B 0,C 180,E1 -2960.961,E2 -2960.961} C_VEL
LIN {X 0,Y 559.05,Z 378.961,A -85,B 0,C 180,E1 -2961.87,E2 -2961.87} C_VEL
LIN {X 0,Y 558.944,Z 386.623,A -85,B 0,C 180,E1 -2962.958,E2 -2962.958} C_VEL
LIN {X 0,Y 558.936,Z 393.679,A -85,B 0,C 180,E1 -2964.227,E2 -2964.227} C_VEL
LIN {X 0,Y 558.826,Z 398.373,A -85,B 0,C 180,E1 -2965.311,E2 -2965.311} C_VEL
LIN {X 0,Y 558.836,Z 401.958,A -85,B 0,C 180,E1 -2966.395,E2 -2966.395} C_VEL
LIN {X 0,Y 558.799,Z 403.807,A -85,B 0,C 180,E1 -2967.116,E2 -2967.116} C_VEL
LIN {X 0,Y 558.745,Z 406.183,A -85,B 0,C 180,E1 -2968.558,E2 -2968.558} C_VEL
LIN {X 0,Y 558.74,Z 407,A -85,B 0,C 180,E1 -2970,E2 -2970} C_VEL
LIN {X 0,Y 558.745,Z 406.184,A -85,B 0,C 180,E1 -2971.441,E2 -2971.441} C_VEL
LIN {X 0,Y 558.799,Z 403.81,A -85,B 0,C 180,E1 -2972.884,E2 -2972.884} C_VEL
LIN {X 0,Y 558.844,Z 400.895,A -85,B 0,C 180,E1 -2973.966,E2 -2973.966} C_VEL
LIN {X 0,Y 558.798,Z 396.948,A -85,B 0,C 180,E1 -2975.051,E2 -2975.051} C_VEL
LIN {X 0,Y 558.922,Z 391.868,A -85,B 0,C 180,E1 -2976.135,E2 -2976.135} C_VEL
LIN {X 0,Y 558.977,Z 385.467,A -85,B 0,C 180,E1 -2977.223,E2 -2977.223} C_VEL
LIN {X 0,Y 559.099,Z 377.478,A -85,B 0,C 180,E1 -2978.312,E2 -2978.312} C_VEL
LIN {X 0,Y 559.195,Z 369.334,A -85,B 0,C 180,E1 -2979.221,E2 -2979.221} C_VEL
LIN {X 0,Y 559.357,Z 359.398,A -85,B 0,C 180,E1 -2980.131,E2 -2980.131} C_VEL
LIN {X 0,Y 559.556,Z 348.398,A -85,B 0,C 180,E1 -2980.937,E2 -2980.937} C_VEL
LIN {X 0,Y 559.672,Z 336.458,A -85,B 0,C 180,E1 -2981.628,E2 -2981.628} C_VEL
LIN {X 0,Y 559.82,Z 324.978,A -85,B 0,C 180,E1 -2982.138,E2 -2982.138} C_VEL
LIN {X 0,Y 559.979,Z 312.177,A -85,B 0,C 180,E1 -2982.549,E2 -2982.549} C_VEL
LIN {X 0,Y 560.079,Z 300.106,A -85,B 0,C 180,E1 -2982.8,E2 -2982.8} C_VEL
LIN {X 0,Y 560.087,Z 198.931,A -85,B 0,C 180,E1 -2984.111,E2 -2984.111} C_VEL
LIN {X 0,Y 559.392,Z 194.063,A -85,B 0,C 180,E1 -2984.204,E2 -2984.204} C_VEL
LIN {X 0,Y 559.632,Z 171.276,A -85,B 0,C 180,E1 -2987.254,E2 -2987.254} C_VEL
LIN {X 0,Y 559.904,Z 148.151,A -85,B 0,C 180,E1 -2990.385,E2 -2990.385} C_VEL
LIN {X 0,Y 560.094,Z 127.036,A -85,B 0,C 180,E1 -2993.282,E2 -2993.282} C_VEL
LIN {X 0,Y 559.947,Z 122.783,A -85,B 0,C 180,E1 -2993.877,E2 -2993.877} C_VEL
LIN {X 0,Y 559.224,Z 118.832,A -85,B 0,C 180,E1 -2994.477,E2 -2994.477} C_VEL
LIN {X 0,Y 559.172,Z 118.832,A -85,B 0,C 180,E1 -2996.902,E2 -2996.902} C_VEL
LIN {X 0,Y 559.15,Z 118.833,A -85,B 0,C 180,E1 -2999.857,E2 -2999.857} C_VEL
LIN {X 0,Y 559.159,Z 118.834,A -85,B 0,C 180,E1 -3002.715,E2 -3002.715} C_VEL
LIN {X 0,Y 559.128,Z 118.833,A -85,B 0,C 180,E1 -3005.324,E2 -3005.324} C_VEL
LIN {X 0,Y 559.136,Z 118.839,A -85,B 0,C 180,E1 -3008.017,E2 -3008.017} C_VEL
LIN {X 0,Y 559.178,Z 118.828,A -85,B 0,C 180,E1 -3010.81,E2 -3010.81} C_VEL
LIN {X 0,Y 559.142,Z 118.835,A -85,B 0,C 180,E1 -3013.733,E2 -3013.733} C_VEL
LIN {X 0,Y 559.146,Z 118.831,A -85,B 0,C 180,E1 -3016.803,E2 -3016.803} C_VEL
LIN {X 0,Y 559.177,Z 118.827,A -85,B 0,C 180,E1 -3019.189,E2 -3019.189} C_VEL
LIN {X 0,Y 559.135,Z 118.841,A -85,B 0,C 180,E1 -3021.982,E2 -3021.982} C_VEL
LIN {X 0,Y 559.131,Z 118.832,A -85,B 0,C 180,E1 -3024.787,E2 -3024.787} C_VEL
LIN {X 0,Y 559.156,Z 118.832,A -85,B 0,C 180,E1 -3027.364,E2 -3027.364} C_VEL
LIN {X 0,Y 559.148,Z 118.832,A -85,B 0,C 180,E1 -3030.142,E2 -3030.142} C_VEL
LIN {X 0,Y 559.168,Z 118.829,A -85,B 0,C 180,E1 -3033.097,E2 -3033.097} C_VEL
LIN {X 0,Y 559.155,Z 118.836,A -85,B 0,C 180,E1 -3035.495,E2 -3035.495} C_VEL
LIN {X 0,Y 559.171,Z 118.826,A -85,B 0,C 180,E1 -3038.624,E2 -3038.624} C_VEL
LIN {X 0,Y 559.167,Z 118.828,A -85,B 0,C 180,E1 -3040.926,E2 -3040.926} C_VEL
LIN {X 0,Y 559.165,Z 118.829,A -85,B 0,C 180,E1 -3043.948,E2 -3043.948} C_VEL
LIN {X 0,Y 559.17,Z 118.827,A -85,B 0,C 180,E1 -3046.184,E2 -3046.184} C_VEL
LIN {X 0,Y 559.195,Z 118.83,A -85,B 0,C 180,E1 -3049.133,E2 -3049.133} C_VEL
LIN {X 0,Y 559.204,Z 118.822,A -85,B 0,C 180,E1 -3052.053,E2 -3052.053} C_VEL
LIN {X 0,Y 559.253,Z 118.823,A -85,B 0,C 180,E1 -3054.953,E2 -3054.953} C_VEL
LIN {X 0,Y 559.255,Z 118.817,A -85,B 0,C 180,E1 -3057.839,E2 -3057.839} C_VEL
LIN {X 0,Y 559.269,Z 118.819,A -85,B 0,C 180,E1 -3060.72,E2 -3060.72} C_VEL
LIN {X 0,Y 559.236,Z 118.827,A -85,B 0,C 180,E1 -3062.881,E2 -3062.881} C_VEL
LIN {X 0,Y 559.232,Z 118.819,A -85,B 0,C 180,E1 -3065.77,E2 -3065.77} C_VEL
LIN {X 0,Y 559.185,Z 118.832,A -85,B 0,C 180,E1 -3068.674,E2 -3068.674} C_VEL
LIN {X 0,Y 559.203,Z 118.823,A -85,B 0,C 180,E1 -3071.6,E2 -3071.6} C_VEL
LIN {X 0,Y 559.198,Z 118.831,A -85,B 0,C 180,E1 -3074.595,E2 -3074.595} C_VEL
LIN {X 0,Y 559.157,Z 118.829,A -85,B 0,C 180,E1 -3077.557,E2 -3077.557} C_VEL
LIN {X 0,Y 559.17,Z 118.828,A -85,B 0,C 180,E1 -3079.837,E2 -3079.837} C_VEL
LIN {X 0,Y 559.14,Z 118.835,A -85,B 0,C 180,E1 -3082.153,E2 -3082.153} C_VEL
LIN {X 0,Y 559.174,Z 118.829,A -85,B 0,C 180,E1 -3085.298,E2 -3085.298} C_VEL
LIN {X 0,Y 559.19,Z 118.827,A -85,B 0,C 180,E1 -3087.712,E2 -3087.712} C_VEL
LIN {X 0,Y 559.143,Z 118.834,A -85,B 0,C 180,E1 -3090.613,E2 -3090.613} C_VEL
LIN {X 0,Y 558.483,Z 118.916,A -85,B 0,C 180,E1 -3091.214,E2 -3091.214} C_VEL
LIN {X 0,Y 555.622,Z 119.278,A -85,B 0,C 180,E1 -3092.191,E2 -3092.191} C_VEL
LIN {X 0,Y 553.209,Z 119.574,A -85,B 0,C 180,E1 -3092.976,E2 -3092.976} C_VEL
LIN {X 0,Y 552.189,Z 119.7,A -85,B 0,C 180,E1 -3093.583,E2 -3093.583} C_VEL
LIN {X 0,Y 552.115,Z 119.711,A -85,B 0,C 180,E1 -3093.788,E2 -3093.788} C_VEL
LIN {X 0,Y 552.181,Z 119.78,A -85,B 0,C 180,E1 -3095.26,E2 -3095.26} C_VEL
LIN {X 0,Y 552.296,Z 127.402,A -85,B 0,C 180,E1 -3096.732,E2 -3096.732} C_VEL
LIN {X 0,Y 552.23,Z 137.63,A -85,B 0,C 180,E1 -3098.7,E2 -3098.7} C_VEL
LIN {X 0,Y 553.415,Z 145.949,A -85,B 0,C 180,E1 -3098.841,E2 -3098.841} C_VEL
LIN {X 0,Y 553.116,Z 243.701,A -85,B 0,C 180,E1 -3100.135,E2 -3100.135} C_VEL
LIN {X 0,Y 552.97,Z 257.124,A -85,B 0,C 180,E1 -3100.465,E2 -3100.465} C_VEL
LIN {X 0,Y 552.84,Z 268.974,A -85,B 0,C 180,E1 -3100.896,E2 -3100.896} C_VEL
LIN {X 0,Y 552.677,Z 281.5,A -85,B 0,C 180,E1 -3101.516,E2 -3101.516} C_VEL
LIN {X 0,Y 552.504,Z 293.101,A -85,B 0,C 180,E1 -3102.267,E2 -3102.267} C_VEL
LIN {X 0,Y 552.313,Z 303.994,A -85,B 0,C 180,E1 -3103.153,E2 -3103.153} C_VEL
LIN {X 0,Y 552.123,Z 313.559,A -85,B 0,C 180,E1 -3104.128,E2 -3104.128} C_VEL
LIN {X 0,Y 551.976,Z 320.885,A -85,B 0,C 180,E1 -3105.036,E2 -3105.036} C_VEL
LIN {X 0,Y 551.88,Z 327.64,A -85,B 0,C 180,E1 -3106.05,E2 -3106.05} C_VEL
LIN {X 0,Y 551.788,Z 334.28,A -85,B 0,C 180,E1 -3107.295,E2 -3107.295} C_VEL
LIN {X 0,Y 551.736,Z 339.26,A -85,B 0,C 180,E1 -3108.519,E2 -3108.519} C_VEL
LIN {X 0,Y 551.672,Z 343.174,A -85,B 0,C 180,E1 -3109.851,E2 -3109.851} C_VEL
LIN {X 0,Y 551.641,Z 345.419,A -85,B 0,C 180,E1 -3111,E2 -3111} C_VEL
LIN {X 0,Y 551.633,Z 346.775,A -85,B 0,C 180,E1 -3112.3,E2 -3112.3} C_VEL
LIN {X 0,Y 551.646,Z 346.933,A -85,B 0,C 180,E1 -3113.381,E2 -3113.381} C_VEL
LIN {X 0,Y 551.668,Z 346.055,A -85,B 0,C 180,E1 -3114.62,E2 -3114.62} C_VEL
LIN {X 0,Y 551.697,Z 343.938,A -85,B 0,C 180,E1 -3115.909,E2 -3115.909} C_VEL
LIN {X 0,Y 551.713,Z 340.44,A -85,B 0,C 180,E1 -3117.218,E2 -3117.218} C_VEL
LIN {X 0,Y 551.79,Z 335.239,A -85,B 0,C 180,E1 -3118.579,E2 -3118.579} C_VEL
LIN {X 0,Y 551.875,Z 329.53,A -85,B 0,C 180,E1 -3119.716,E2 -3119.716} C_VEL
LIN {X 0,Y 551.973,Z 322.317,A -85,B 0,C 180,E1 -3120.855,E2 -3120.855} C_VEL
LIN {X 0,Y 552.086,Z 314.08,A -85,B 0,C 180,E1 -3121.901,E2 -3121.901} C_VEL
LIN {X 0,Y 552.285,Z 304.462,A -85,B 0,C 180,E1 -3122.891,E2 -3122.891} C_VEL
LIN {X 0,Y 552.438,Z 293.919,A -85,B 0,C 180,E1 -3123.763,E2 -3123.763} C_VEL
LIN {X 0,Y 552.647,Z 282.003,A -85,B 0,C 180,E1 -3124.542,E2 -3124.542} C_VEL
LIN {X 0,Y 552.824,Z 270.004,A -85,B 0,C 180,E1 -3125.15,E2 -3125.15} C_VEL
LIN {X 0,Y 553,Z 256.932,A -85,B 0,C 180,E1 -3125.629,E2 -3125.629} C_VEL
LIN {X 0,Y 553.121,Z 243.455,A -85,B 0,C 180,E1 -3125.959,E2 -3125.959} C_VEL
LIN {X 0,Y 553.306,Z 143.574,A -85,B 0,C 180,E1 -3127.281,E2 -3127.281} C_VEL
LIN {X 0,Y 552.184,Z 137.486,A -85,B 0,C 180,E1 -3127.405,E2 -3127.405} C_VEL
LIN {X 0,Y 552.321,Z 122.577,A -85,B 0,C 180,E1 -3130.324,E2 -3130.324} C_VEL
LIN {X 0,Y 552.149,Z 119.708,A -85,B 0,C 180,E1 -3130.916,E2 -3130.916} C_VEL
LIN {X 0,Y 552.111,Z 119.716,A -85,B 0,C 180,E1 -3133.737,E2 -3133.737} C_VEL
LIN {X 0,Y 552.133,Z 119.709,A -85,B 0,C 180,E1 -3136.005,E2 -3136.005} C_VEL
LIN {X 0,Y 552.163,Z 119.701,A -85,B 0,C 180,E1 -3138.994,E2 -3138.994} C_VEL
LIN {X 0,Y 552.154,Z 119.704,A -85,B 0,C 180,E1 -3141.952,E2 -3141.952} C_VEL
LIN {X 0,Y 552.228,Z 119.693,A -85,B 0,C 180,E1 -3144.889,E2 -3144.889} C_VEL
LIN {X 0,Y 552.228,Z 119.695,A -85,B 0,C 180,E1 -3147.812,E2 -3147.812} C_VEL
LIN {X 0,Y 552.237,Z 119.692,A -85,B 0,C 180,E1 -3150.729,E2 -3150.729} C_VEL
LIN {X 0,Y 552.2,Z 119.699,A -85,B 0,C 180,E1 -3152.918,E2 -3152.918} C_VEL
LIN {X 0,Y 552.201,Z 119.696,A -85,B 0,C 180,E1 -3155.844,E2 -3155.844} C_VEL
LIN {X 0,Y 552.142,Z 119.707,A -85,B 0,C 180,E1 -3158.786,E2 -3158.786} C_VEL
LIN {X 0,Y 552.163,Z 119.701,A -85,B 0,C 180,E1 -3161.75,E2 -3161.75} C_VEL
LIN {X 0,Y 552.137,Z 119.709,A -85,B 0,C 180,E1 -3164.748,E2 -3164.748} C_VEL
LIN {X 0,Y 552.097,Z 119.708,A -85,B 0,C 180,E1 -3167.789,E2 -3167.789} C_VEL
LIN {X 0,Y 552.126,Z 119.705,A -85,B 0,C 180,E1 -3170.101,E2 -3170.101} C_VEL
LIN {X 0,Y 552.092,Z 119.713,A -85,B 0,C 180,E1 -3172.451,E2 -3172.451} C_VEL
LIN {X 0,Y 552.155,Z 119.702,A -85,B 0,C 180,E1 -3175.35,E2 -3175.35} C_VEL
LIN {X 0,Y 552.109,Z 119.709,A -85,B 0,C 180,E1 -3178.098,E2 -3178.098} C_VEL
LIN {X 0,Y 552.1,Z 119.717,A -85,B 0,C 180,E1 -3180.609,E2 -3180.609} C_VEL
LIN {X 0,Y 552.106,Z 119.708,A -85,B 0,C 180,E1 -3183.186,E2 -3183.186} C_VEL
LIN {X 0,Y 552.084,Z 119.711,A -85,B 0,C 180,E1 -3185.844,E2 -3185.844} C_VEL
LIN {X 0,Y 552.116,Z 119.712,A -85,B 0,C 180,E1 -3188.589,E2 -3188.589} C_VEL
LIN {X 0,Y 552.129,Z 119.704,A -85,B 0,C 180,E1 -3191.445,E2 -3191.445} C_VEL
LIN {X 0,Y 552.094,Z 119.713,A -85,B 0,C 180,E1 -3194.532,E2 -3194.532} C_VEL
LIN {X 0,Y 552.128,Z 119.706,A -85,B 0,C 180,E1 -3197.585,E2 -3197.585} C_VEL
LIN {X 0,Y 552.131,Z 119.708,A -85,B 0,C 180,E1 -3200.473,E2 -3200.473} C_VEL
LIN {X 0,Y 552.109,Z 119.707,A -85,B 0,C 180,E1 -3203.316,E2 -3203.316} C_VEL
LIN {X 0,Y 552.126,Z 119.714,A -85,B 0,C 180,E1 -3205.939,E2 -3205.939} C_VEL
LIN {X 0,Y 552.117,Z 119.707,A -85,B 0,C 180,E1 -3208.541,E2 -3208.541} C_VEL
LIN {X 0,Y 552.123,Z 119.709,A -85,B 0,C 180,E1 -3211.438,E2 -3211.438} C_VEL
LIN {X 0,Y 552.128,Z 119.706,A -85,B 0,C 180,E1 -3214.356,E2 -3214.356} C_VEL
LIN {X 0,Y 552.095,Z 119.708,A -85,B 0,C 180,E1 -3216.758,E2 -3216.758} C_VEL
LIN {X 0,Y 552.119,Z 119.708,A -85,B 0,C 180,E1 -3219.12,E2 -3219.12} C_VEL
LIN {X 0,Y 552.124,Z 119.712,A -85,B 0,C 180,E1 -3221.444,E2 -3221.444} C_VEL
LIN {X 0,Y 552.115,Z 119.712,A -85,B 0,C 180,E1 -3223.737,E2 -3223.737} C_VEL
LIN {X 0,Y 552.134,Z 119.705,A -85,B 0,C 180,E1 -3226.005,E2 -3226.005} C_VEL
LIN {X 0,Y 552.162,Z 119.704,A -85,B 0,C 180,E1 -3228.994,E2 -3228.994} C_VEL
LIN {X 0,Y 552.158,Z 119.702,A -85,B 0,C 180,E1 -3231.952,E2 -3231.952} C_VEL
LIN {X 0,Y 552.229,Z 119.696,A -85,B 0,C 180,E1 -3234.889,E2 -3234.889} C_VEL
LIN {X 0,Y 552.226,Z 119.693,A -85,B 0,C 180,E1 -3237.812,E2 -3237.812} C_VEL
LIN {X 0,Y 552.239,Z 119.694,A -85,B 0,C 180,E1 -3240.729,E2 -3240.729} C_VEL
LIN {X 0,Y 552.203,Z 119.703,A -85,B 0,C 180,E1 -3242.918,E2 -3242.918} C_VEL
LIN {X 0,Y 552.202,Z 119.695,A -85,B 0,C 180,E1 -3245.844,E2 -3245.844} C_VEL
LIN {X 0,Y 552.156,Z 119.709,A -85,B 0,C 180,E1 -3248.786,E2 -3248.786} C_VEL
LIN {X 0,Y 552.162,Z 119.7,A -85,B 0,C 180,E1 -3251.751,E2 -3251.751} C_VEL
LIN {X 0,Y 552.136,Z 119.713,A -85,B 0,C 180,E1 -3254.749,E2 -3254.749} C_VEL
LIN {X 0,Y 552.11,Z 119.707,A -85,B 0,C 180,E1 -3257.789,E2 -3257.789} C_VEL
LIN {X 0,Y 552.13,Z 119.706,A -85,B 0,C 180,E1 -3260.101,E2 -3260.101} C_VEL
LIN {X 0,Y 552.092,Z 119.717,A -85,B 0,C 180,E1 -3262.451,E2 -3262.451} C_VEL
LIN {X 0,Y 552.155,Z 119.701,A -85,B 0,C 180,E1 -3265.351,E2 -3265.351} C_VEL
LIN {X 0,Y 552.109,Z 119.711,A -85,B 0,C 180,E1 -3268.099,E2 -3268.099} C_VEL
LIN {X 0,Y 552.104,Z 119.712,A -85,B 0,C 180,E1 -3270.609,E2 -3270.609} C_VEL
LIN {X 0,Y 552.115,Z 119.706,A -85,B 0,C 180,E1 -3273.186,E2 -3273.186} C_VEL
LIN {X 0,Y 552.085,Z 119.713,A -85,B 0,C 180,E1 -3275.844,E2 -3275.844} C_VEL
LIN {X 0,Y 552.126,Z 119.704,A -85,B 0,C 180,E1 -3279.062,E2 -3279.062} C_VEL
LIN {X 0,Y 552.14,Z 119.704,A -85,B 0,C 180,E1 -3281.444,E2 -3281.444} C_VEL
LIN {X 0,Y 552.096,Z 119.71,A -85,B 0,C 180,E1 -3284.532,E2 -3284.532} C_VEL
LIN {X 0,Y 552.132,Z 119.708,A -85,B 0,C 180,E1 -3287.585,E2 -3287.585} C_VEL
LIN {X 0,Y 552.135,Z 119.705,A -85,B 0,C 180,E1 -3290.474,E2 -3290.474} C_VEL
LIN {X 0,Y 552.108,Z 119.71,A -85,B 0,C 180,E1 -3293.317,E2 -3293.317} C_VEL
LIN {X 0,Y 552.128,Z 119.71,A -85,B 0,C 180,E1 -3295.939,E2 -3295.939} C_VEL
LIN {X 0,Y 552.121,Z 119.705,A -85,B 0,C 180,E1 -3298.541,E2 -3298.541} C_VEL
LIN {X 0,Y 552.127,Z 119.713,A -85,B 0,C 180,E1 -3301.438,E2 -3301.438} C_VEL
LIN {X 0,Y 552.132,Z 119.708,A -85,B 0,C 180,E1 -3304.356,E2 -3304.356} C_VEL
LIN {X 0,Y 552.219,Z 119.834,A -85,B 0,C 180,E1 -3305.317,E2 -3305.317} C_VEL
LIN {X 0,Y 553.243,Z 126.249,A -85,B 0,C 180,E1 -3306.279,E2 -3306.279} C_VEL
LIN {X 0,Y 552.979,Z 142.54,A -85,B 0,C 180,E1 -3308.568,E2 -3308.568} C_VEL
LIN {X 0,Y 552.802,Z 160.648,A -85,B 0,C 180,E1 -3311.083,E2 -3311.083} C_VEL
LIN {X 0,Y 552.538,Z 180.084,A -85,B 0,C 180,E1 -3313.75,E2 -3313.75} C_VEL
LIN {X 0,Y 552.375,Z 193.753,A -85,B 0,C 180,E1 -3315.611,E2 -3315.611} C_VEL
LIN {X 0,Y 553.365,Z 201.611,A -85,B 0,C 180,E1 -3315.755,E2 -3315.755} C_VEL
LIN {X 0,Y 553.133,Z 302.434,A -85,B 0,C 180,E1 -3317.083,E2 -3317.083} C_VEL
LIN {X 0,Y 552.953,Z 315.789,A -85,B 0,C 180,E1 -3317.405,E2 -3317.405} C_VEL
LIN {X 0,Y 552.818,Z 329.143,A -85,B 0,C 180,E1 -3317.891,E2 -3317.891} C_VEL
LIN {X 0,Y 552.65,Z 340.758,A -85,B 0,C 180,E1 -3318.47,E2 -3318.47} C_VEL
LIN {X 0,Y 552.439,Z 351.999,A -85,B 0,C 180,E1 -3319.185,E2 -3319.185} C_VEL
LIN {X 0,Y 552.274,Z 362.491,A -85,B 0,C 180,E1 -3320.015,E2 -3320.015} C_VEL
LIN {X 0,Y 552.126,Z 371.071,A -85,B 0,C 180,E1 -3320.845,E2 -3320.845} C_VEL
LIN {X 0,Y 552.013,Z 378.961,A -85,B 0,C 180,E1 -3321.765,E2 -3321.765} C_VEL
LIN {X 0,Y 551.89,Z 386.621,A -85,B 0,C 180,E1 -3322.868,E2 -3322.868} C_VEL
LIN {X 0,Y 551.867,Z 393.679,A -85,B 0,C 180,E1 -3324.153,E2 -3324.153} C_VEL
LIN {X 0,Y 551.725,Z 398.373,A -85,B 0,C 180,E1 -3325.251,E2 -3325.251} C_VEL
LIN {X 0,Y 551.75,Z 401.958,A -85,B 0,C 180,E1 -3326.348,E2 -3326.348} C_VEL
LIN {X 0,Y 551.723,Z 403.807,A -85,B 0,C 180,E1 -3327.079,E2 -3327.079} C_VEL
LIN {X 0,Y 551.645,Z 406.182,A -85,B 0,C 180,E1 -3328.54,E2 -3328.54} C_VEL
LIN {X 0,Y 551.64,Z 407,A -85,B 0,C 180,E1 -3330,E2 -3330} C_VEL
LIN {X 0,Y 551.645,Z 406.183,A -85,B 0,C 180,E1 -3331.46,E2 -3331.46} C_VEL
LIN {X 0,Y 551.723,Z 403.81,A -85,B 0,C 180,E1 -3332.921,E2 -3332.921} C_VEL
LIN {X 0,Y 551.764,Z 400.895,A -85,B 0,C 180,E1 -3334.017,E2 -3334.017} C_VEL
LIN {X 0,Y 551.723,Z 396.948,A -85,B 0,C 180,E1 -3335.116,E2 -3335.116} C_VEL
LIN {X 0,Y 551.803,Z 391.189,A -85,B 0,C 180,E1 -3336.341,E2 -3336.341} C_VEL
LIN {X 0,Y 551.926,Z 384.235,A -85,B 0,C 180,E1 -3337.5,E2 -3337.5} C_VEL
LIN {X 0,Y 552.082,Z 375.987,A -85,B 0,C 180,E1 -3338.602,E2 -3338.602} C_VEL
LIN {X 0,Y 552.2,Z 367.466,A -85,B 0,C 180,E1 -3339.524,E2 -3339.524} C_VEL
LIN {X 0,Y 552.396,Z 356.927,A -85,B 0,C 180,E1 -3340.445,E2 -3340.445} C_VEL
LIN {X 0,Y 552.555,Z 346.035,A -85,B 0,C 180,E1 -3341.214,E2 -3341.214} C_VEL
LIN {X 0,Y 552.723,Z 335.074,A -85,B 0,C 180,E1 -3341.831,E2 -3341.831} C_VEL
LIN {X 0,Y 552.9,Z 323.346,A -85,B 0,C 180,E1 -3342.34,E2 -3342.34} C_VEL
LIN {X 0,Y 553.027,Z 310.752,A -85,B 0,C 180,E1 -3342.733,E2 -3342.733} C_VEL
LIN {X 0,Y 553.158,Z 297.977,A -85,B 0,C 180,E1 -3342.986,E2 -3342.986} C_VEL
LIN {X 0,Y 553.236,Z 200.028,A -85,B 0,C 180,E1 -3344.267,E2 -3344.267} C_VEL
LIN {X 0,Y 552.357,Z 193.561,A -85,B 0,C 180,E1 -3344.399,E2 -3344.399} C_VEL
LIN {X 0,Y 552.613,Z 172.587,A -85,B 0,C 180,E1 -3347.241,E2 -3347.241} C_VEL
LIN {X 0,Y 552.859,Z 151.911,A -85,B 0,C 180,E1 -3350.073,E2 -3350.073} C_VEL
LIN {X 0,Y 553.139,Z 129.395,A -85,B 0,C 180,E1 -3353.196,E2 -3353.196} C_VEL
LIN {X 0,Y 552.912,Z 123.723,A -85,B 0,C 180,E1 -3354,E2 -3354} C_VEL
LIN {X 0,Y 552.165,Z 119.711,A -85,B 0,C 180,E1 -3354.61,E2 -3354.61} C_VEL
LIN {X 0,Y 552.132,Z 119.706,A -85,B 0,C 180,E1 -3357.273,E2 -3357.273} C_VEL
LIN {X 0,Y 552.118,Z 119.712,A -85,B 0,C 180,E1 -3360.05,E2 -3360.05} C_VEL
LIN {X 0,Y 552.117,Z 119.709,A -85,B 0,C 180,E1 -3362.846,E2 -3362.846} C_VEL
LIN {X 0,Y 552.078,Z 119.712,A -85,B 0,C 180,E1 -3365.439,E2 -3365.439} C_VEL
LIN {X 0,Y 552.099,Z 119.714,A -85,B 0,C 180,E1 -3367.886,E2 -3367.886} C_VEL
LIN {X 0,Y 552.143,Z 119.708,A -85,B 0,C 180,E1 -3370.478,E2 -3370.478} C_VEL
LIN {X 0,Y 552.119,Z 119.708,A -85,B 0,C 180,E1 -3373.484,E2 -3373.484} C_VEL
LIN {X 0,Y 552.106,Z 119.71,A -85,B 0,C 180,E1 -3376.576,E2 -3376.576} C_VEL
LIN {X 0,Y 552.142,Z 119.706,A -85,B 0,C 180,E1 -3379.522,E2 -3379.522} C_VEL
LIN {X 0,Y 552.093,Z 119.712,A -85,B 0,C 180,E1 -3382.336,E2 -3382.336} C_VEL
LIN {X 0,Y 552.083,Z 119.71,A -85,B 0,C 180,E1 -3385.051,E2 -3385.051} C_VEL
LIN {X 0,Y 552.116,Z 119.713,A -85,B 0,C 180,E1 -3387.681,E2 -3387.681} C_VEL
LIN {X 0,Y 552.111,Z 119.708,A -85,B 0,C 180,E1 -3390.235,E2 -3390.235} C_VEL
LIN {X 0,Y 552.137,Z 119.704,A -85,B 0,C 180,E1 -3393,E2 -3393} C_VEL
LIN {X 0,Y 552.112,Z 119.708,A -85,B 0,C 180,E1 -3395.161,E2 -3395.161} C_VEL
LIN {X 0,Y 552.124,Z 119.705,A -85,B 0,C 180,E1 -3398.337,E2 -3398.337} C_VEL
LIN {X 0,Y 552.155,Z 119.7,A -85,B 0,C 180,E1 -3400.674,E2 -3400.674} C_VEL
LIN {X 0,Y 552.115,Z 119.71,A -85,B 0,C 180,E1 -3403.737,E2 -3403.737} C_VEL
LIN {X 0,Y 552.134,Z 119.705,A -85,B 0,C 180,E1 -3406.004,E2 -3406.004} C_VEL
LIN {X 0,Y 552.162,Z 119.704,A -85,B 0,C 180,E1 -3408.993,E2 -3408.993} C_VEL
LIN {X 0,Y 552.158,Z 119.7,A -85,B 0,C 180,E1 -3411.951,E2 -3411.951} C_VEL
LIN {X 0,Y 552.229,Z 119.697,A -85,B 0,C 180,E1 -3414.889,E2 -3414.889} C_VEL
LIN {X 0,Y 552.226,Z 119.693,A -85,B 0,C 180,E1 -3417.812,E2 -3417.812} C_VEL
LIN {X 0,Y 552.239,Z 119.694,A -85,B 0,C 180,E1 -3420.729,E2 -3420.729} C_VEL
LIN {X 0,Y 552.203,Z 119.703,A -85,B 0,C 180,E1 -3422.918,E2 -3422.918} C_VEL
LIN {X 0,Y 552.201,Z 119.695,A -85,B 0,C 180,E1 -3425.844,E2 -3425.844} C_VEL
LIN {X 0,Y 552.156,Z 119.71,A -85,B 0,C 180,E1 -3428.786,E2 -3428.786} C_VEL
LIN {X 0,Y 552.161,Z 119.7,A -85,B 0,C 180,E1 -3431.75,E2 -3431.75} C_VEL
LIN {X 0,Y 552.135,Z 119.713,A -85,B 0,C 180,E1 -3434.748,E2 -3434.748} C_VEL
LIN {X 0,Y 552.108,Z 119.707,A -85,B 0,C 180,E1 -3437.788,E2 -3437.788} C_VEL
LIN {X 0,Y 552.129,Z 119.707,A -85,B 0,C 180,E1 -3440.101,E2 -3440.101} C_VEL
LIN {X 0,Y 552.091,Z 119.718,A -85,B 0,C 180,E1 -3442.451,E2 -3442.451} C_VEL
LIN {X 0,Y 552.153,Z 119.703,A -85,B 0,C 180,E1 -3445.35,E2 -3445.35} C_VEL
LIN {X 0,Y 552.124,Z 119.711,A -85,B 0,C 180,E1 -3448.097,E2 -3448.097} C_VEL
LIN {X 0,Y 552.105,Z 119.714,A -85,B 0,C 180,E1 -3450.609,E2 -3450.609} C_VEL
LIN {X 0,Y 552.121,Z 119.707,A -85,B 0,C 180,E1 -3453.185,E2 -3453.185} C_VEL
LIN {X 0,Y 552.115,Z 119.711,A -85,B 0,C 180,E1 -3453.788,E2 -3453.788} C_VEL
LIN {X 0,Y 551.474,Z 119.833,A -85,B 0,C 180,E1 -3454.201,E2 -3454.201} C_VEL
LIN {X 0,Y 548.729,Z 120.626,A -85,B 0,C 180,E1 -3454.845,E2 -3454.845} C_VEL
LIN {X 0,Y 545.977,Z 122.412,A -85,B 0,C 180,E1 -3455.469,E2 -3455.469} C_VEL
LIN {X 0,Y 545.328,Z 124.105,A -85,B 0,C 180,E1 -3455.845,E2 -3455.845} C_VEL
LIN {X 0,Y 545.28,Z 138.022,A -85,B 0,C 180,E1 -3458.513,E2 -3458.513} C_VEL
LIN {X 0,Y 546.552,Z 146.096,A -85,B 0,C 180,E1 -3458.657,E2 -3458.657} C_VEL
LIN {X 0,Y 546.205,Z 244.326,A -85,B 0,C 180,E1 -3459.977,E2 -3459.977} C_VEL
LIN {X 0,Y 546.043,Z 257.608,A -85,B 0,C 180,E1 -3460.308,E2 -3460.308} C_VEL
LIN {X 0,Y 545.912,Z 269.534,A -85,B 0,C 180,E1 -3460.75,E2 -3460.75} C_VEL
LIN {X 0,Y 545.753,Z 281.34,A -85,B 0,C 180,E1 -3461.338,E2 -3461.338} C_VEL
LIN {X 0,Y 545.577,Z 292.464,A -85,B 0,C 180,E1 -3462.056,E2 -3462.056} C_VEL
LIN {X 0,Y 545.358,Z 302.631,A -85,B 0,C 180,E1 -3462.871,E2 -3462.871} C_VEL
LIN {X 0,Y 545.151,Z 311.925,A -85,B 0,C 180,E1 -3463.785,E2 -3463.785} C_VEL
LIN {X 0,Y 544.98,Z 320.487,A -85,B 0,C 180,E1 -3464.825,E2 -3464.825} C_VEL
LIN {X 0,Y 544.834,Z 327.365,A -85,B 0,C 180,E1 -3465.848,E2 -3465.848} C_VEL
LIN {X 0,Y 544.745,Z 334.238,A -85,B 0,C 180,E1 -3467.132,E2 -3467.132} C_VEL
LIN {X 0,Y 544.662,Z 339.62,A -85,B 0,C 180,E1 -3468.452,E2 -3468.452} C_VEL
LIN {X 0,Y 544.605,Z 343.582,A -85,B 0,C 180,E1 -3469.817,E2 -3469.817} C_VEL
LIN {X 0,Y 544.567,Z 345.51,A -85,B 0,C 180,E1 -3470.775,E2 -3470.775} C_VEL
LIN {X 0,Y 544.544,Z 346.919,A -85,B 0,C 180,E1 -3471.932,E2 -3471.932} C_VEL
LIN {X 0,Y 544.56,Z 347.353,A -85,B 0,C 180,E1 -3473.145,E2 -3473.145} C_VEL
LIN {X 0,Y 544.567,Z 346.585,A -85,B 0,C 180,E1 -3474.497,E2 -3474.497} C_VEL
LIN {X 0,Y 544.588,Z 344.832,A -85,B 0,C 180,E1 -3475.683,E2 -3475.683} C_VEL
LIN {X 0,Y 544.651,Z 341.625,A -85,B 0,C 180,E1 -3477.007,E2 -3477.007} C_VEL
LIN {X 0,Y 544.717,Z 336.779,A -85,B 0,C 180,E1 -3478.379,E2 -3478.379} C_VEL
LIN {X 0,Y 544.799,Z 331.093,A -85,B 0,C 180,E1 -3479.58,E2 -3479.58} C_VEL
LIN {X 0,Y 544.931,Z 323.587,A -85,B 0,C 180,E1 -3480.826,E2 -3480.826} C_VEL
LIN {X 0,Y 545.078,Z 315.202,A -85,B 0,C 180,E1 -3481.926,E2 -3481.926} C_VEL
LIN {X 0,Y 545.242,Z 306.308,A -85,B 0,C 180,E1 -3482.874,E2 -3482.874} C_VEL
LIN {X 0,Y 545.476,Z 295.42,A -85,B 0,C 180,E1 -3483.815,E2 -3483.815} C_VEL
LIN {X 0,Y 545.648,Z 284.523,A -85,B 0,C 180,E1 -3484.56,E2 -3484.56} C_VEL
LIN {X 0,Y 545.857,Z 272.297,A -85,B 0,C 180,E1 -3485.213,E2 -3485.213} C_VEL
LIN {X 0,Y 546.043,Z 260.736,A -85,B 0,C 180,E1 -3485.678,E2 -3485.678} C_VEL
LIN {X 0,Y 546.192,Z 248.545,A -85,B 0,C 180,E1 -3486.025,E2 -3486.025} C_VEL
LIN {X 0,Y 546.298,Z 233.068,A -85,B 0,C 180,E1 -3486.28,E2 -3486.28} C_VEL
LIN {X 0,Y 546.464,Z 144.478,A -85,B 0,C 180,E1 -3487.455,E2 -3487.455} C_VEL
LIN {X 0,Y 545.187,Z 137.734,A -85,B 0,C 180,E1 -3487.599,E2 -3487.599} C_VEL
LIN {X 0,Y 545.339,Z 123.365,A -85,B 0,C 180,E1 -3490.423,E2 -3490.423} C_VEL
LIN {X 0,Y 545.105,Z 120.586,A -85,B 0,C 180,E1 -3491.001,E2 -3491.001} C_VEL
LIN {X 0,Y 545.063,Z 120.592,A -85,B 0,C 180,E1 -3493.521,E2 -3493.521} C_VEL
LIN {X 0,Y 545.094,Z 120.589,A -85,B 0,C 180,E1 -3495.82,E2 -3495.82} C_VEL
LIN {X 0,Y 545.118,Z 120.578,A -85,B 0,C 180,E1 -3498.849,E2 -3498.849} C_VEL
LIN {X 0,Y 545.125,Z 120.581,A -85,B 0,C 180,E1 -3501.847,E2 -3501.847} C_VEL
LIN {X 0,Y 545.204,Z 120.568,A -85,B 0,C 180,E1 -3504.823,E2 -3504.823} C_VEL
LIN {X 0,Y 545.199,Z 120.571,A -85,B 0,C 180,E1 -3507.784,E2 -3507.784} C_VEL
LIN {X 0,Y 545.208,Z 120.568,A -85,B 0,C 180,E1 -3510.739,E2 -3510.739} C_VEL
LIN {X 0,Y 545.167,Z 120.576,A -85,B 0,C 180,E1 -3512.956,E2 -3512.956} C_VEL
LIN {X 0,Y 545.171,Z 120.572,A -85,B 0,C 180,E1 -3515.919,E2 -3515.919} C_VEL
LIN {X 0,Y 545.102,Z 120.585,A -85,B 0,C 180,E1 -3518.9,E2 -3518.9} C_VEL
LIN {X 0,Y 545.135,Z 120.575,A -85,B 0,C 180,E1 -3521.904,E2 -3521.904} C_VEL
LIN {X 0,Y 545.085,Z 120.591,A -85,B 0,C 180,E1 -3524.944,E2 -3524.944} C_VEL
LIN {X 0,Y 545.069,Z 120.584,A -85,B 0,C 180,E1 -3528.026,E2 -3528.026} C_VEL
LIN {X 0,Y 545.092,Z 120.583,A -85,B 0,C 180,E1 -3530.372,E2 -3530.372} C_VEL
LIN {X 0,Y 545.08,Z 120.583,A -85,B 0,C 180,E1 -3533.559,E2 -3533.559} C_VEL
LIN {X 0,Y 545.078,Z 120.583,A -85,B 0,C 180,E1 -3536,E2 -3536} C_VEL
LIN {X 0,Y 545.088,Z 120.589,A -85,B 0,C 180,E1 -3538.748,E2 -3538.748} C_VEL
LIN {X 0,Y 545.057,Z 120.585,A -85,B 0,C 180,E1 -3541.679,E2 -3541.679} C_VEL
LIN {X 0,Y 545.058,Z 120.593,A -85,B 0,C 180,E1 -3544.565,E2 -3544.565} C_VEL
LIN {X 0,Y 545.037,Z 120.588,A -85,B 0,C 180,E1 -3547.304,E2 -3547.304} C_VEL
LIN {X 0,Y 545.065,Z 120.59,A -85,B 0,C 180,E1 -3550.142,E2 -3550.142} C_VEL
LIN {X 0,Y 545.077,Z 120.583,A -85,B 0,C 180,E1 -3553.106,E2 -3553.106} C_VEL
LIN {X 0,Y 545.055,Z 120.594,A -85,B 0,C 180,E1 -3556.225,E2 -3556.225} C_VEL
LIN {X 0,Y 545.09,Z 120.581,A -85,B 0,C 180,E1 -3558.886,E2 -3558.886} C_VEL
LIN {X 0,Y 545.052,Z 120.59,A -85,B 0,C 180,E1 -3561.763,E2 -3561.763} C_VEL
LIN {X 0,Y 545.049,Z 120.588,A -85,B 0,C 180,E1 -3564.533,E2 -3564.533} C_VEL
LIN {X 0,Y 545.067,Z 120.585,A -85,B 0,C 180,E1 -3567.212,E2 -3567.212} C_VEL
LIN {X 0,Y 545.101,Z 120.589,A -85,B 0,C 180,E1 -3569.813,E2 -3569.813} C_VEL
LIN {X 0,Y 545.085,Z 120.582,A -85,B 0,C 180,E1 -3572.828,E2 -3572.828} C_VEL
LIN {X 0,Y 545.047,Z 120.595,A -85,B 0,C 180,E1 -3575.631,E2 -3575.631} C_VEL
LIN {X 0,Y 545.064,Z 120.585,A -85,B 0,C 180,E1 -3578.837,E2 -3578.837} C_VEL
LIN {X 0,Y 545.078,Z 120.586,A -85,B 0,C 180,E1 -3581.196,E2 -3581.196} C_VEL
LIN {X 0,Y 545.072,Z 120.593,A -85,B 0,C 180,E1 -3583.521,E2 -3583.521} C_VEL
LIN {X 0,Y 545.093,Z 120.584,A -85,B 0,C 180,E1 -3585.82,E2 -3585.82} C_VEL
LIN {X 0,Y 545.117,Z 120.58,A -85,B 0,C 180,E1 -3588.849,E2 -3588.849} C_VEL
LIN {X 0,Y 545.129,Z 120.578,A -85,B 0,C 180,E1 -3591.847,E2 -3591.847} C_VEL
LIN {X 0,Y 545.205,Z 120.57,A -85,B 0,C 180,E1 -3594.823,E2 -3594.823} C_VEL
LIN {X 0,Y 545.197,Z 120.569,A -85,B 0,C 180,E1 -3597.784,E2 -3597.784} C_VEL
LIN {X 0,Y 545.21,Z 120.57,A -85,B 0,C 180,E1 -3600.739,E2 -3600.739} C_VEL
LIN {X 0,Y 545.17,Z 120.579,A -85,B 0,C 180,E1 -3602.956,E2 -3602.956} C_VEL
LIN {X 0,Y 545.172,Z 120.571,A -85,B 0,C 180,E1 -3605.92,E2 -3605.92} C_VEL
LIN {X 0,Y 545.116,Z 120.587,A -85,B 0,C 180,E1 -3608.9,E2 -3608.9} C_VEL
LIN {X 0,Y 545.134,Z 120.575,A -85,B 0,C 180,E1 -3611.904,E2 -3611.904} C_VEL
LIN {X 0,Y 545.085,Z 120.588,A -85,B 0,C 180,E1 -3614.944,E2 -3614.944} C_VEL
LIN {X 0,Y 545.078,Z 120.584,A -85,B 0,C 180,E1 -3618.026,E2 -3618.026} C_VEL
LIN {X 0,Y 545.095,Z 120.586,A -85,B 0,C 180,E1 -3620.372,E2 -3620.372} C_VEL
LIN {X 0,Y 545.08,Z 120.582,A -85,B 0,C 180,E1 -3623.56,E2 -3623.56} C_VEL
LIN {X 0,Y 545.08,Z 120.585,A -85,B 0,C 180,E1 -3626.001,E2 -3626.001} C_VEL
LIN {X 0,Y 545.089,Z 120.585,A -85,B 0,C 180,E1 -3628.748,E2 -3628.748} C_VEL
LIN {X 0,Y 545.057,Z 120.586,A -85,B 0,C 180,E1 -3631.679,E2 -3631.679} C_VEL
LIN {X 0,Y 545.062,Z 120.589,A -85,B 0,C 180,E1 -3634.565,E2 -3634.565} C_VEL
LIN {X 0,Y 545.037,Z 120.588,A -85,B 0,C 180,E1 -3637.304,E2 -3637.304} C_VEL
LIN {X 0,Y 545.093,Z 120.59,A -85,B 0,C 180,E1 -3640.14,E2 -3640.14} C_VEL
LIN {X 0,Y 545.079,Z 120.582,A -85,B 0,C 180,E1 -3643.107,E2 -3643.107} C_VEL
LIN {X 0,Y 545.068,Z 120.589,A -85,B 0,C 180,E1 -3646.225,E2 -3646.225} C_VEL
LIN {X 0,Y 545.103,Z 120.579,A -85,B 0,C 180,E1 -3648.888,E2 -3648.888} C_VEL
LIN {X 0,Y 545.056,Z 120.594,A -85,B 0,C 180,E1 -3651.763,E2 -3651.763} C_VEL
LIN {X 0,Y 545.037,Z 120.588,A -85,B 0,C 180,E1 -3654.532,E2 -3654.532} C_VEL
LIN {X 0,Y 545.071,Z 120.586,A -85,B 0,C 180,E1 -3657.212,E2 -3657.212} C_VEL
LIN {X 0,Y 545.066,Z 120.592,A -85,B 0,C 180,E1 -3659.811,E2 -3659.811} C_VEL
LIN {X 0,Y 545.083,Z 120.584,A -85,B 0,C 180,E1 -3662.344,E2 -3662.344} C_VEL
LIN {X 0,Y 545.159,Z 120.719,A -85,B 0,C 180,E1 -3665.154,E2 -3665.154} C_VEL
LIN {X 0,Y 546.323,Z 127.931,A -85,B 0,C 180,E1 -3666.25,E2 -3666.25} C_VEL
LIN {X 0,Y 546.011,Z 146.365,A -85,B 0,C 180,E1 -3668.875,E2 -3668.875} C_VEL
LIN {X 0,Y 545.672,Z 168.629,A -85,B 0,C 180,E1 -3671.995,E2 -3671.995} C_VEL
LIN {X 0,Y 545.367,Z 188.029,A -85,B 0,C 180,E1 -3674.682,E2 -3674.682} C_VEL
LIN {X 0,Y 545.334,Z 193.542,A -85,B 0,C 180,E1 -3675.439,E2 -3675.439} C_VEL
LIN {X 0,Y 546.469,Z 202.131,A -85,B 0,C 180,E1 -3675.585,E2 -3675.585} C_VEL
LIN {X 0,Y 546.226,Z 301.908,A -85,B 0,C 180,E1 -3676.917,E2 -3676.917} C_VEL
LIN {X 0,Y 546.028,Z 315.317,A -85,B 0,C 180,E1 -3677.243,E2 -3677.243} C_VEL
LIN {X 0,Y 545.857,Z 327.564,A -85,B 0,C 180,E1 -3677.687,E2 -3677.687} C_VEL
LIN {X 0,Y 545.693,Z 338.823,A -85,B 0,C 180,E1 -3678.235,E2 -3678.235} C_VEL
LIN {X 0,Y 545.485,Z 350.281,A -85,B 0,C 180,E1 -3678.951,E2 -3678.951} C_VEL
LIN {X 0,Y 545.248,Z 361.001,A -85,B 0,C 180,E1 -3679.792,E2 -3679.792} C_VEL
LIN {X 0,Y 545.085,Z 370.665,A -85,B 0,C 180,E1 -3680.725,E2 -3680.725} C_VEL
LIN {X 0,Y 544.947,Z 378.589,A -85,B 0,C 180,E1 -3681.658,E2 -3681.658} C_VEL
LIN {X 0,Y 544.824,Z 386.33,A -85,B 0,C 180,E1 -3682.775,E2 -3682.775} C_VEL
LIN {X 0,Y 544.777,Z 393.467,A -85,B 0,C 180,E1 -3684.076,E2 -3684.076} C_VEL
LIN {X 0,Y 544.629,Z 398.209,A -85,B 0,C 180,E1 -3685.189,E2 -3685.189} C_VEL
LIN {X 0,Y 544.669,Z 401.841,A -85,B 0,C 180,E1 -3686.301,E2 -3686.301} C_VEL
LIN {X 0,Y 544.65,Z 403.711,A -85,B 0,C 180,E1 -3687.041,E2 -3687.041} C_VEL
LIN {X 0,Y 544.546,Z 406.111,A -85,B 0,C 180,E1 -3688.521,E2 -3688.521} C_VEL
LIN {X 0,Y 544.542,Z 406.722,A -85,B 0,C 180,E1 -3689.26,E2 -3689.26} C_VEL
LIN {X 0,Y 544.541,Z 406.94,A -85,B 0,C 180,E1 -3690,E2 -3690} C_VEL
LIN {X 0,Y 544.542,Z 406.722,A -85,B 0,C 180,E1 -3690.739,E2 -3690.739} C_VEL
LIN {X 0,Y 544.572,Z 405.113,A -85,B 0,C 180,E1 -3692.219,E2 -3692.219} C_VEL
LIN {X 0,Y 544.65,Z 403.714,A -85,B 0,C 180,E1 -3692.959,E2 -3692.959} C_VEL
LIN {X 0,Y 544.684,Z 400.763,A -85,B 0,C 180,E1 -3694.069,E2 -3694.069} C_VEL
LIN {X 0,Y 544.653,Z 396.764,A -85,B 0,C 180,E1 -3695.182,E2 -3695.182} C_VEL
LIN {X 0,Y 544.709,Z 391.456,A -85,B 0,C 180,E1 -3696.328,E2 -3696.328} C_VEL
LIN {X 0,Y 544.836,Z 385.147,A -85,B 0,C 180,E1 -3697.411,E2 -3697.411} C_VEL
LIN {X 0,Y 544.969,Z 377.071,A -85,B 0,C 180,E1 -3698.529,E2 -3698.529} C_VEL
LIN {X 0,Y 545.114,Z 368.841,A -85,B 0,C 180,E1 -3699.461,E2 -3699.461} C_VEL
LIN {X 0,Y 545.343,Z 358.809,A -85,B 0,C 180,E1 -3700.394,E2 -3700.394} C_VEL
LIN {X 0,Y 545.53,Z 347.898,A -85,B 0,C 180,E1 -3701.208,E2 -3701.208} C_VEL
LIN {X 0,Y 545.704,Z 336.376,A -85,B 0,C 180,E1 -3701.891,E2 -3701.891} C_VEL
LIN {X 0,Y 545.923,Z 324.077,A -85,B 0,C 180,E1 -3702.453,E2 -3702.453} C_VEL
LIN {X 0,Y 546.067,Z 311.125,A -85,B 0,C 180,E1 -3702.874,E2 -3702.874} C_VEL
LIN {X 0,Y 546.244,Z 297.357,A -85,B 0,C 180,E1 -3703.154,E2 -3703.154} C_VEL
LIN {X 0,Y 546.351,Z 200.738,A -85,B 0,C 180,E1 -3704.435,E2 -3704.435} C_VEL
LIN {X 0,Y 545.292,Z 193.141,A -85,B 0,C 180,E1 -3704.588,E2 -3704.588} C_VEL
LIN {X 0,Y 545.607,Z 171.222,A -85,B 0,C 180,E1 -3707.598,E2 -3707.598} C_VEL
LIN {X 0,Y 545.912,Z 150.063,A -85,B 0,C 180,E1 -3710.537,E2 -3710.537} C_VEL
LIN {X 0,Y 546.199,Z 128.929,A -85,B 0,C 180,E1 -3713.508,E2 -3713.508} C_VEL
LIN {X 0,Y 545.933,Z 124.891,A -85,B 0,C 180,E1 -3714.093,E2 -3714.093} C_VEL
LIN {X 0,Y 545.126,Z 120.587,A -85,B 0,C 180,E1 -3714.772,E2 -3714.772} C_VEL
LIN {X 0,Y 545.083,Z 120.585,A -85,B 0,C 180,E1 -3717.656,E2 -3717.656} C_VEL
LIN {X 0,Y 545.079,Z 120.591,A -85,B 0,C 180,E1 -3720.246,E2 -3720.246} C_VEL
LIN {X 0,Y 545.081,Z 120.584,A -85,B 0,C 180,E1 -3723.062,E2 -3723.062} C_VEL
LIN {X 0,Y 545.035,Z 120.591,A -85,B 0,C 180,E1 -3725.673,E2 -3725.673} C_VEL
LIN {X 0,Y 545.056,Z 120.596,A -85,B 0,C 180,E1 -3728.237,E2 -3728.237} C_VEL
LIN {X 0,Y 545.102,Z 120.581,A -85,B 0,C 180,E1 -3731.112,E2 -3731.112} C_VEL
LIN {X 0,Y 545.059,Z 120.595,A -85,B 0,C 180,E1 -3734.129,E2 -3734.129} C_VEL
LIN {X 0,Y 545.078,Z 120.584,A -85,B 0,C 180,E1 -3736.893,E2 -3736.893} C_VEL
LIN {X 0,Y 545.093,Z 120.589,A -85,B 0,C 180,E1 -3739.86,E2 -3739.86} C_VEL
LIN {X 0,Y 545.07,Z 120.584,A -85,B 0,C 180,E1 -3743.074,E2 -3743.074} C_VEL
LIN {X 0,Y 545.065,Z 120.586,A -85,B 0,C 180,E1 -3746.328,E2 -3746.328} C_VEL
LIN {X 0,Y 545.066,Z 120.585,A -85,B 0,C 180,E1 -3748.952,E2 -3748.952} C_VEL
LIN {X 0,Y 545.1,Z 120.585,A -85,B 0,C 180,E1 -3751.507,E2 -3751.507} C_VEL
LIN {X 0,Y 545.094,Z 120.58,A -85,B 0,C 180,E1 -3754.491,E2 -3754.491} C_VEL
LIN {X 0,Y 545.035,Z 120.591,A -85,B 0,C 180,E1 -3757.242,E2 -3757.242} C_VEL
LIN {X 0,Y 545.119,Z 120.576,A -85,B 0,C 180,E1 -3760.415,E2 -3760.415} C_VEL
LIN {X 0,Y 545.072,Z 120.59,A -85,B 0,C 180,E1 -3763.521,E2 -3763.521} C_VEL
LIN {X 0,Y 545.093,Z 120.584,A -85,B 0,C 180,E1 -3765.82,E2 -3765.82} C_VEL
LIN {X 0,Y 545.117,Z 120.58,A -85,B 0,C 180,E1 -3768.849,E2 -3768.849} C_VEL
LIN {X 0,Y 545.128,Z 120.577,A -85,B 0,C 180,E1 -3771.847,E2 -3771.847} C_VEL
LIN {X 0,Y 545.205,Z 120.571,A -85,B 0,C 180,E1 -3774.823,E2 -3774.823} C_VEL
LIN {X 0,Y 545.197,Z 120.569,A -85,B 0,C 180,E1 -3777.784,E2 -3777.784} C_VEL
LIN {X 0,Y 545.21,Z 120.57,A -85,B 0,C 180,E1 -3780.738,E2 -3780.738} C_VEL
LIN {X 0,Y 545.169,Z 120.579,A -85,B 0,C 180,E1 -3782.956,E2 -3782.956} C_VEL
LIN {X 0,Y 545.171,Z 120.57,A -85,B 0,C 180,E1 -3785.919,E2 -3785.919} C_VEL
LIN {X 0,Y 545.115,Z 120.586,A -85,B 0,C 180,E1 -3788.9,E2 -3788.9} C_VEL
LIN {X 0,Y 545.133,Z 120.576,A -85,B 0,C 180,E1 -3791.904,E2 -3791.904} C_VEL
LIN {X 0,Y 545.083,Z 120.588,A -85,B 0,C 180,E1 -3794.943,E2 -3794.943} C_VEL
LIN {X 0,Y 545.077,Z 120.585,A -85,B 0,C 180,E1 -3798.026,E2 -3798.026} C_VEL
LIN {X 0,Y 545.093,Z 120.587,A -85,B 0,C 180,E1 -3800.372,E2 -3800.372} C_VEL
LIN {X 0,Y 545.079,Z 120.585,A -85,B 0,C 180,E1 -3803.559,E2 -3803.559} C_VEL
LIN {X 0,Y 545.078,Z 120.587,A -85,B 0,C 180,E1 -3806,E2 -3806} C_VEL
LIN {X 0,Y 545.088,Z 120.587,A -85,B 0,C 180,E1 -3808.749,E2 -3808.749} C_VEL
LIN {X 0,Y 545.076,Z 120.586,A -85,B 0,C 180,E1 -3811.683,E2 -3811.683} C_VEL
LIN {X 0,Y 545.094,Z 120.59,A -85,B 0,C 180,E1 -3814.562,E2 -3814.562} C_VEL
LIN {X 0,Y 545.157,Z 120.638,A -85,B 0,C 180,E1 -3815.176,E2 -3815.176} C_VEL
LIN {X 0,Y 545.328,Z 124.105,A -85,B 0,C 180,E1 -3815.845,E2 -3815.845} C_VEL
LIN {X 0,Y 544.659,Z 126.093,A -85,B 0,C 180,E1 -3816.2,E2 -3816.2} C_VEL
LIN {X 0,Y 541.812,Z 129.442,A -85,B 0,C 180,E1 -3816.739,E2 -3816.739} C_VEL
LIN {X 0,Y 538.946,Z 132.794,A -85,B 0,C 180,E1 -3817.283,E2 -3817.283} C_VEL
LIN {X 0,Y 538.262,Z 134.783,A -85,B 0,C 180,E1 -3817.644,E2 -3817.644} C_VEL
LIN {X 0,Y 538.289,Z 138.499,A -85,B 0,C 180,E1 -3818.321,E2 -3818.321} C_VEL
LIN {X 0,Y 539.621,Z 145.692,A -85,B 0,C 180,E1 -3818.458,E2 -3818.458} C_VEL
LIN {X 0,Y 539.318,Z 245.134,A -85,B 0,C 180,E1 -3819.819,E2 -3819.819} C_VEL
LIN {X 0,Y 539.127,Z 258.811,A -85,B 0,C 180,E1 -3820.171,E2 -3820.171} C_VEL
LIN {X 0,Y 538.98,Z 270.636,A -85,B 0,C 180,E1 -3820.623,E2 -3820.623} C_VEL
LIN {X 0,Y 538.778,Z 282.722,A -85,B 0,C 180,E1 -3821.247,E2 -3821.247} C_VEL
LIN {X 0,Y 538.591,Z 293.797,A -85,B 0,C 180,E1 -3821.984,E2 -3821.984} C_VEL
LIN {X 0,Y 538.359,Z 304.644,A -85,B 0,C 180,E1 -3822.886,E2 -3822.886} C_VEL
LIN {X 0,Y 538.119,Z 314.697,A -85,B 0,C 180,E1 -3823.94,E2 -3823.94} C_VEL
LIN {X 0,Y 537.91,Z 321.976,A -85,B 0,C 180,E1 -3824.872,E2 -3824.872} C_VEL
LIN {X 0,Y 537.772,Z 328.92,A -85,B 0,C 180,E1 -3825.954,E2 -3825.954} C_VEL
LIN {X 0,Y 537.687,Z 335.227,A -85,B 0,C 180,E1 -3827.182,E2 -3827.182} C_VEL
LIN {X 0,Y 537.632,Z 339.29,A -85,B 0,C 180,E1 -3828.189,E2 -3828.189} C_VEL
LIN {X 0,Y 537.57,Z 342.816,A -85,B 0,C 180,E1 -3829.312,E2 -3829.312} C_VEL
LIN {X 0,Y 537.494,Z 345.448,A -85,B 0,C 180,E1 -3830.484,E2 -3830.484} C_VEL
LIN {X 0,Y 537.467,Z 347.093,A -85,B 0,C 180,E1 -3831.681,E2 -3831.681} C_VEL
LIN {X 0,Y 537.489,Z 347.754,A -85,B 0,C 180,E1 -3833.024,E2 -3833.024} C_VEL
LIN {X 0,Y 537.481,Z 347.305,A -85,B 0,C 180,E1 -3834.164,E2 -3834.164} C_VEL
LIN {X 0,Y 537.491,Z 345.699,A -85,B 0,C 180,E1 -3835.463,E2 -3835.463} C_VEL
LIN {X 0,Y 537.57,Z 342.745,A -85,B 0,C 180,E1 -3836.794,E2 -3836.794} C_VEL
LIN {X 0,Y 537.659,Z 338.239,A -85,B 0,C 180,E1 -3838.173,E2 -3838.173} C_VEL
LIN {X 0,Y 537.729,Z 333.066,A -85,B 0,C 180,E1 -3839.355,E2 -3839.355} C_VEL
LIN {X 0,Y 537.828,Z 327.066,A -85,B 0,C 180,E1 -3840.443,E2 -3840.443} C_VEL
LIN {X 0,Y 537.993,Z 319.699,A -85,B 0,C 180,E1 -3841.523,E2 -3841.523} C_VEL
LIN {X 0,Y 538.17,Z 310.373,A -85,B 0,C 180,E1 -3842.625,E2 -3842.625} C_VEL
LIN {X 0,Y 538.399,Z 300.728,A -85,B 0,C 180,E1 -3843.548,E2 -3843.548} C_VEL
LIN {X 0,Y 538.619,Z 289.626,A -85,B 0,C 180,E1 -3844.399,E2 -3844.399} C_VEL
LIN {X 0,Y 538.888,Z 277.495,A -85,B 0,C 180,E1 -3845.128,E2 -3845.128} C_VEL
LIN {X 0,Y 539.038,Z 266.378,A -85,B 0,C 180,E1 -3845.643,E2 -3845.643} C_VEL
LIN {X 0,Y 539.221,Z 253.64,A -85,B 0,C 180,E1 -3846.071,E2 -3846.071} C_VEL
LIN {X 0,Y 539.358,Z 240.227,A -85,B 0,C 180,E1 -3846.354,E2 -3846.354} C_VEL
LIN {X 0,Y 539.554,Z 145.069,A -85,B 0,C 180,E1 -3847.64,E2 -3847.64} C_VEL
LIN {X 0,Y 538.172,Z 138.052,A -85,B 0,C 180,E1 -3847.79,E2 -3847.79} C_VEL
LIN {X 0,Y 538.321,Z 124.016,A -85,B 0,C 180,E1 -3850.554,E2 -3850.554} C_VEL
LIN {X 0,Y 538.055,Z 121.464,A -85,B 0,C 180,E1 -3851.089,E2 -3851.089} C_VEL
LIN {X 0,Y 538.019,Z 121.467,A -85,B 0,C 180,E1 -3854.079,E2 -3854.079} C_VEL
LIN {X 0,Y 538.027,Z 121.463,A -85,B 0,C 180,E1 -3856.401,E2 -3856.401} C_VEL
LIN {X 0,Y 538.078,Z 121.454,A -85,B 0,C 180,E1 -3858.702,E2 -3858.702} C_VEL
LIN {X 0,Y 538.082,Z 121.46,A -85,B 0,C 180,E1 -3861.74,E2 -3861.74} C_VEL
LIN {X 0,Y 538.162,Z 121.445,A -85,B 0,C 180,E1 -3864.755,E2 -3864.755} C_VEL
LIN {X 0,Y 538.171,Z 121.447,A -85,B 0,C 180,E1 -3867.755,E2 -3867.755} C_VEL
LIN {X 0,Y 538.179,Z 121.444,A -85,B 0,C 180,E1 -3870.748,E2 -3870.748} C_VEL
LIN {X 0,Y 538.135,Z 121.452,A -85,B 0,C 180,E1 -3872.994,E2 -3872.994} C_VEL
LIN {X 0,Y 538.121,Z 121.449,A -85,B 0,C 180,E1 -3875.997,E2 -3875.997} C_VEL
LIN {X 0,Y 538.055,Z 121.465,A -85,B 0,C 180,E1 -3879.018,E2 -3879.018} C_VEL
LIN {X 0,Y 538.083,Z 121.454,A -85,B 0,C 180,E1 -3882.062,E2 -3882.062} C_VEL
LIN {X 0,Y 538.045,Z 121.465,A -85,B 0,C 180,E1 -3885.144,E2 -3885.144} C_VEL
LIN {X 0,Y 538.024,Z 121.463,A -85,B 0,C 180,E1 -3888.27,E2 -3888.27} C_VEL
LIN {X 0,Y 538.037,Z 121.466,A -85,B 0,C 180,E1 -3890.651,E2 -3890.651} C_VEL
LIN {X 0,Y 538.003,Z 121.464,A -85,B 0,C 180,E1 -3893.888,E2 -3893.888} C_VEL
LIN {X 0,Y 538.041,Z 121.463,A -85,B 0,C 180,E1 -3896.367,E2 -3896.367} C_VEL
LIN {X 0,Y 538.029,Z 121.465,A -85,B 0,C 180,E1 -3898.933,E2 -3898.933} C_VEL
LIN {X 0,Y 538.009,Z 121.464,A -85,B 0,C 180,E1 -3901.887,E2 -3901.887} C_VEL
LIN {X 0,Y 538.008,Z 121.47,A -85,B 0,C 180,E1 -3904.617,E2 -3904.617} C_VEL
LIN {X 0,Y 538.005,Z 121.464,A -85,B 0,C 180,E1 -3907.17,E2 -3907.17} C_VEL
LIN {X 0,Y 538.021,Z 121.463,A -85,B 0,C 180,E1 -3909.797,E2 -3909.797} C_VEL
LIN {X 0,Y 538.018,Z 121.464,A -85,B 0,C 180,E1 -3912.786,E2 -3912.786} C_VEL
LIN {X 0,Y 538.03,Z 121.46,A -85,B 0,C 180,E1 -3915.14,E2 -3915.14} C_VEL
LIN {X 0,Y 538.033,Z 121.468,A -85,B 0,C 180,E1 -3918.227,E2 -3918.227} C_VEL
LIN {X 0,Y 538.014,Z 121.463,A -85,B 0,C 180,E1 -3921.17,E2 -3921.17} C_VEL
LIN {X 0,Y 538.021,Z 121.47,A -85,B 0,C 180,E1 -3924.084,E2 -3924.084} C_VEL
LIN {X 0,Y 538.028,Z 121.461,A -85,B 0,C 180,E1 -3926.727,E2 -3926.727} C_VEL
LIN {X 0,Y 538.037,Z 121.464,A -85,B 0,C 180,E1 -3929.554,E2 -3929.554} C_VEL
LIN {X 0,Y 538.038,Z 121.466,A -85,B 0,C 180,E1 -3931.95,E2 -3931.95} C_VEL
LIN {X 0,Y 538.069,Z 121.456,A -85,B 0,C 180,E1 -3934.467,E2 -3934.467} C_VEL
LIN {X 0,Y 537.991,Z 121.473,A -85,B 0,C 180,E1 -3937.738,E2 -3937.738} C_VEL
LIN {X 0,Y 538.078,Z 121.456,A -85,B 0,C 180,E1 -3940.148,E2 -3940.148} C_VEL
LIN {X 0,Y 538.023,Z 121.467,A -85,B 0,C 180,E1 -3943.299,E2 -3943.299} C_VEL
LIN {X 0,Y 538.062,Z 121.463,A -85,B 0,C 180,E1 -3945.631,E2 -3945.631} C_VEL
LIN {X 0,Y 538.076,Z 121.456,A -85,B 0,C 180,E1 -3948.702,E2 -3948.702} C_VEL
LIN {X 0,Y 538.086,Z 121.457,A -85,B 0,C 180,E1 -3951.74,E2 -3951.74} C_VEL
LIN {X 0,Y 538.163,Z 121.446,A -85,B 0,C 180,E1 -3954.755,E2 -3954.755} C_VEL
LIN {X 0,Y 538.169,Z 121.445,A -85,B 0,C 180,E1 -3957.755,E2 -3957.755} C_VEL
LIN {X 0,Y 538.18,Z 121.446,A -85,B 0,C 180,E1 -3960.748,E2 -3960.748} C_VEL
LIN {X 0,Y 538.136,Z 121.456,A -85,B 0,C 180,E1 -3962.995,E2 -3962.995} C_VEL
LIN {X 0,Y 538.121,Z 121.449,A -85,B 0,C 180,E1 -3965.997,E2 -3965.997} C_VEL
LIN {X 0,Y 538.067,Z 121.463,A -85,B 0,C 180,E1 -3969.018,E2 -3969.018} C_VEL
LIN {X 0,Y 538.082,Z 121.455,A -85,B 0,C 180,E1 -3972.063,E2 -3972.063} C_VEL
LIN {X 0,Y 538.044,Z 121.462,A -85,B 0,C 180,E1 -3975.144,E2 -3975.144} C_VEL
LIN {X 0,Y 538.031,Z 121.464,A -85,B 0,C 180,E1 -3978.27,E2 -3978.27} C_VEL
LIN {X 0,Y 538.039,Z 121.468,A -85,B 0,C 180,E1 -3980.652,E2 -3980.652} C_VEL
LIN {X 0,Y 538.003,Z 121.465,A -85,B 0,C 180,E1 -3983.889,E2 -3983.889} C_VEL
LIN {X 0,Y 538.042,Z 121.467,A -85,B 0,C 180,E1 -3986.367,E2 -3986.367} C_VEL
LIN {X 0,Y 538.03,Z 121.462,A -85,B 0,C 180,E1 -3988.934,E2 -3988.934} C_VEL
LIN {X 0,Y 538.01,Z 121.466,A -85,B 0,C 180,E1 -3991.888,E2 -3991.888} C_VEL
LIN {X 0,Y 538.012,Z 121.466,A -85,B 0,C 180,E1 -3994.618,E2 -3994.618} C_VEL
LIN {X 0,Y 538.005,Z 121.464,A -85,B 0,C 180,E1 -3997.17,E2 -3997.17} C_VEL
LIN {X 0,Y 538.055,Z 121.462,A -85,B 0,C 180,E1 -3999.794,E2 -3999.794} C_VEL
LIN {X 0,Y 538.02,Z 121.462,A -85,B 0,C 180,E1 -4002.786,E2 -4002.786} C_VEL
LIN {X 0,Y 538.032,Z 121.46,A -85,B 0,C 180,E1 -4005.141,E2 -4005.141} C_VEL
LIN {X 0,Y 538.042,Z 121.463,A -85,B 0,C 180,E1 -4008.228,E2 -4008.228} C_VEL
LIN {X 0,Y 538.06,Z 121.458,A -85,B 0,C 180,E1 -4010.412,E2 -4010.412} C_VEL
LIN {X 0,Y 538.026,Z 121.462,A -85,B 0,C 180,E1 -4013.067,E2 -4013.067} C_VEL
LIN {X 0,Y 538.02,Z 121.47,A -85,B 0,C 180,E1 -4015.827,E2 -4015.827} C_VEL
LIN {X 0,Y 538.011,Z 121.463,A -85,B 0,C 180,E1 -4018.499,E2 -4018.499} C_VEL
LIN {X 0,Y 538.062,Z 121.461,A -85,B 0,C 180,E1 -4021.1,E2 -4021.1} C_VEL
LIN {X 0,Y 538.044,Z 121.468,A -85,B 0,C 180,E1 -4023.634,E2 -4023.634} C_VEL
LIN {X 0,Y 538.129,Z 121.601,A -85,B 0,C 180,E1 -4024.987,E2 -4024.987} C_VEL
LIN {X 0,Y 539.402,Z 129.321,A -85,B 0,C 180,E1 -4026.178,E2 -4026.178} C_VEL
LIN {X 0,Y 539.023,Z 148.794,A -85,B 0,C 180,E1 -4028.989,E2 -4028.989} C_VEL
LIN {X 0,Y 538.663,Z 171.857,A -85,B 0,C 180,E1 -4032.259,E2 -4032.259} C_VEL
LIN {X 0,Y 538.307,Z 193.084,A -85,B 0,C 180,E1 -4035.237,E2 -4035.237} C_VEL
LIN {X 0,Y 539.593,Z 203.32,A -85,B 0,C 180,E1 -4035.418,E2 -4035.418} C_VEL
LIN {X 0,Y 539.282,Z 302.546,A -85,B 0,C 180,E1 -4036.769,E2 -4036.769} C_VEL
LIN {X 0,Y 539.063,Z 316.37,A -85,B 0,C 180,E1 -4037.123,E2 -4037.123} C_VEL
LIN {X 0,Y 538.878,Z 329.291,A -85,B 0,C 180,E1 -4037.621,E2 -4037.621} C_VEL
LIN {X 0,Y 538.615,Z 341.055,A -85,B 0,C 180,E1 -4038.235,E2 -4038.235} C_VEL
LIN {X 0,Y 538.409,Z 352.459,A -85,B 0,C 180,E1 -4038.994,E2 -4038.994} C_VEL
LIN {X 0,Y 538.16,Z 362.719,A -85,B 0,C 180,E1 -4039.846,E2 -4039.846} C_VEL
LIN {X 0,Y 537.99,Z 371.95,A -85,B 0,C 180,E1 -4040.792,E2 -4040.792} C_VEL
LIN {X 0,Y 537.815,Z 380.943,A -85,B 0,C 180,E1 -4041.925,E2 -4041.925} C_VEL
LIN {X 0,Y 537.679,Z 388.183,A -85,B 0,C 180,E1 -4043.056,E2 -4043.056} C_VEL
LIN {X 0,Y 537.657,Z 394.782,A -85,B 0,C 180,E1 -4044.374,E2 -4044.374} C_VEL
LIN {X 0,Y 537.553,Z 399.142,A -85,B 0,C 180,E1 -4045.501,E2 -4045.501} C_VEL
LIN {X 0,Y 537.591,Z 401.454,A -85,B 0,C 180,E1 -4046.252,E2 -4046.252} C_VEL
LIN {X 0,Y 537.58,Z 403.326,A -85,B 0,C 180,E1 -4047.002,E2 -4047.002} C_VEL
LIN {X 0,Y 537.455,Z 405.725,A -85,B 0,C 180,E1 -4048.501,E2 -4048.501} C_VEL
LIN {X 0,Y 537.452,Z 406.336,A -85,B 0,C 180,E1 -4049.251,E2 -4049.251} C_VEL
LIN {X 0,Y 537.453,Z 406.552,A -85,B 0,C 180,E1 -4050,E2 -4050} C_VEL
LIN {X 0,Y 537.452,Z 406.334,A -85,B 0,C 180,E1 -4050.749,E2 -4050.749} C_VEL
LIN {X 0,Y 537.49,Z 404.722,A -85,B 0,C 180,E1 -4052.248,E2 -4052.248} C_VEL
LIN {X 0,Y 537.58,Z 403.32,A -85,B 0,C 180,E1 -4052.998,E2 -4052.998} C_VEL
LIN {X 0,Y 537.603,Z 400.364,A -85,B 0,C 180,E1 -4054.123,E2 -4054.123} C_VEL
LIN {X 0,Y 537.587,Z 396.36,A -85,B 0,C 180,E1 -4055.251,E2 -4055.251} C_VEL
LIN {X 0,Y 537.644,Z 390.278,A -85,B 0,C 180,E1 -4056.554,E2 -4056.554} C_VEL
LIN {X 0,Y 537.784,Z 383.485,A -85,B 0,C 180,E1 -4057.698,E2 -4057.698} C_VEL
LIN {X 0,Y 537.929,Z 375.142,A -85,B 0,C 180,E1 -4058.83,E2 -4058.83} C_VEL
LIN {X 0,Y 538.082,Z 366.589,A -85,B 0,C 180,E1 -4059.776,E2 -4059.776} C_VEL
LIN {X 0,Y 538.335,Z 356.029,A -85,B 0,C 180,E1 -4060.721,E2 -4060.721} C_VEL
LIN {X 0,Y 538.539,Z 344.872,A -85,B 0,C 180,E1 -4061.526,E2 -4061.526} C_VEL
LIN {X 0,Y 538.767,Z 334.123,A -85,B 0,C 180,E1 -4062.142,E2 -4062.142} C_VEL
LIN {X 0,Y 538.976,Z 322.333,A -85,B 0,C 180,E1 -4062.664,E2 -4062.664} C_VEL
LIN {X 0,Y 539.162,Z 309.665,A -85,B 0,C 180,E1 -4063.066,E2 -4063.066} C_VEL
LIN {X 0,Y 539.327,Z 296.738,A -85,B 0,C 180,E1 -4063.326,E2 -4063.326} C_VEL
LIN {X 0,Y 539.461,Z 201.245,A -85,B 0,C 180,E1 -4064.611,E2 -4064.611} C_VEL
LIN {X 0,Y 538.261,Z 192.702,A -85,B 0,C 180,E1 -4064.785,E2 -4064.785} C_VEL
LIN {X 0,Y 538.58,Z 171.648,A -85,B 0,C 180,E1 -4067.713,E2 -4067.713} C_VEL
LIN {X 0,Y 538.917,Z 151.017,A -85,B 0,C 180,E1 -4070.616,E2 -4070.616} C_VEL
LIN {X 0,Y 539.271,Z 129.889,A -85,B 0,C 180,E1 -4073.625,E2 -4073.625} C_VEL
LIN {X 0,Y 538.777,Z 125.041,A -85,B 0,C 180,E1 -4074.344,E2 -4074.344} C_VEL
LIN {X 0,Y 538.093,Z 121.462,A -85,B 0,C 180,E1 -4074.911,E2 -4074.911} C_VEL
LIN {X 0,Y 538.042,Z 121.465,A -85,B 0,C 180,E1 -4078.05,E2 -4078.05} C_VEL
LIN {X 0,Y 538.022,Z 121.468,A -85,B 0,C 180,E1 -4080.627,E2 -4080.627} C_VEL
LIN {X 0,Y 538.047,Z 121.46,A -85,B 0,C 180,E1 -4083.282,E2 -4083.282} C_VEL
LIN {X 0,Y 537.995,Z 121.471,A -85,B 0,C 180,E1 -4086.004,E2 -4086.004} C_VEL
LIN {X 0,Y 538.017,Z 121.465,A -85,B 0,C 180,E1 -4088.83,E2 -4088.83} C_VEL
LIN {X 0,Y 538.079,Z 121.457,A -85,B 0,C 180,E1 -4090.773,E2 -4090.773} C_VEL
LIN {X 0,Y 538.03,Z 121.47,A -85,B 0,C 180,E1 -4094.074,E2 -4094.074} C_VEL
LIN {X 0,Y 538.026,Z 121.462,A -85,B 0,C 180,E1 -4097.012,E2 -4097.012} C_VEL
LIN {X 0,Y 538.079,Z 121.456,A -85,B 0,C 180,E1 -4099.249,E2 -4099.249} C_VEL
LIN {X 0,Y 537.993,Z 121.472,A -85,B 0,C 180,E1 -4102.122,E2 -4102.122} C_VEL
LIN {X 0,Y 537.997,Z 121.465,A -85,B 0,C 180,E1 -4104.915,E2 -4104.915} C_VEL
LIN {X 0,Y 538.018,Z 121.468,A -85,B 0,C 180,E1 -4107.617,E2 -4107.617} C_VEL
LIN {X 0,Y 538.017,Z 121.463,A -85,B 0,C 180,E1 -4110.239,E2 -4110.239} C_VEL
LIN {X 0,Y 538.056,Z 121.457,A -85,B 0,C 180,E1 -4112.796,E2 -4112.796} C_VEL
LIN {X 0,Y 538.026,Z 121.464,A -85,B 0,C 180,E1 -4115.291,E2 -4115.291} C_VEL
LIN {X 0,Y 538.014,Z 121.464,A -85,B 0,C 180,E1 -4118.042,E2 -4118.042} C_VEL
LIN {X 0,Y 538.036,Z 121.46,A -85,B 0,C 180,E1 -4120.94,E2 -4120.94} C_VEL
LIN {X 0,Y 538.024,Z 121.468,A -85,B 0,C 180,E1 -4123.299,E2 -4123.299} C_VEL
LIN {X 0,Y 538.062,Z 121.462,A -85,B 0,C 180,E1 -4125.63,E2 -4125.63} C_VEL
LIN {X 0,Y 538.076,Z 121.455,A -85,B 0,C 180,E1 -4128.701,E2 -4128.701} C_VEL
LIN {X 0,Y 538.085,Z 121.455,A -85,B 0,C 180,E1 -4131.739,E2 -4131.739} C_VEL
LIN {X 0,Y 538.163,Z 121.448,A -85,B 0,C 180,E1 -4134.755,E2 -4134.755} C_VEL
LIN {X 0,Y 538.169,Z 121.445,A -85,B 0,C 180,E1 -4137.755,E2 -4137.755} C_VEL
LIN {X 0,Y 538.18,Z 121.446,A -85,B 0,C 180,E1 -4140.748,E2 -4140.748} C_VEL
LIN {X 0,Y 538.136,Z 121.455,A -85,B 0,C 180,E1 -4142.994,E2 -4142.994} C_VEL
LIN {X 0,Y 538.12,Z 121.449,A -85,B 0,C 180,E1 -4145.997,E2 -4145.997} C_VEL
LIN {X 0,Y 538.067,Z 121.463,A -85,B 0,C 180,E1 -4149.018,E2 -4149.018} C_VEL
LIN {X 0,Y 538.081,Z 121.455,A -85,B 0,C 180,E1 -4152.062,E2 -4152.062} C_VEL
LIN {X 0,Y 538.043,Z 121.463,A -85,B 0,C 180,E1 -4155.144,E2 -4155.144} C_VEL
LIN {X 0,Y 538.029,Z 121.465,A -85,B 0,C 180,E1 -4158.27,E2 -4158.27} C_VEL
LIN {X 0,Y 538.037,Z 121.469,A -85,B 0,C 180,E1 -4160.651,E2 -4160.651} C_VEL
LIN {X 0,Y 538.002,Z 121.468,A -85,B 0,C 180,E1 -4163.888,E2 -4163.888} C_VEL
LIN {X 0,Y 538.041,Z 121.468,A -85,B 0,C 180,E1 -4166.367,E2 -4166.367} C_VEL
LIN {X 0,Y 538.029,Z 121.464,A -85,B 0,C 180,E1 -4168.934,E2 -4168.934} C_VEL
LIN {X 0,Y 538.026,Z 121.466,A -85,B 0,C 180,E1 -4171.89,E2 -4171.89} C_VEL
LIN {X 0,Y 538.085,Z 121.47,A -85,B 0,C 180,E1 -4175.078,E2 -4175.078} C_VEL
LIN {X 0,Y 538.348,Z 128.55,A -85,B 0,C 180,E1 -4176.441,E2 -4176.441} C_VEL
LIN {X 0,Y 538.262,Z 134.783,A -85,B 0,C 180,E1 -4177.644,E2 -4177.644} C_VEL
LIN {X 0,Y 537.87,Z 137.21,A -85,B 0,C 180,E1 -4177.943,E2 -4177.943} C_VEL
LIN {X 0,Y 536.983,Z 140.376,A -85,B 0,C 180,E1 -4178.145,E2 -4178.145} C_VEL
LIN {X 0,Y 535.315,Z 145.861,A -85,B 0,C 180,E1 -4178.316,E2 -4178.316} C_VEL
LIN {X 0,Y 533.108,Z 156.196,A -85,B 0,C 180,E1 -4178.416,E2 -4178.416} C_VEL
LIN {X 0,Y 532.783,Z 164.756,A -85,B 0,C 180,E1 -4178.523,E2 -4178.523} C_VEL
LIN {X 0,Y 532.429,Z 245.616,A -85,B 0,C 180,E1 -4179.649,E2 -4179.649} C_VEL
LIN {X 0,Y 532.221,Z 259.28,A -85,B 0,C 180,E1 -4180.007,E2 -4180.007} C_VEL
LIN {X 0,Y 532.062,Z 270.944,A -85,B 0,C 180,E1 -4180.458,E2 -4180.458} C_VEL
LIN {X 0,Y 531.868,Z 282.459,A -85,B 0,C 180,E1 -4181.054,E2 -4181.054} C_VEL
LIN {X 0,Y 531.671,Z 292.992,A -85,B 0,C 180,E1 -4181.751,E2 -4181.751} C_VEL
LIN {X 0,Y 531.386,Z 302.747,A -85,B 0,C 180,E1 -4182.545,E2 -4182.545} C_VEL
LIN {X 0,Y 531.155,Z 312.077,A -85,B 0,C 180,E1 -4183.475,E2 -4183.475} C_VEL
LIN {X 0,Y 530.958,Z 320.849,A -85,B 0,C 180,E1 -4184.55,E2 -4184.55} C_VEL
LIN {X 0,Y 530.773,Z 328.057,A -85,B 0,C 180,E1 -4185.644,E2 -4185.644} C_VEL
LIN {X 0,Y 530.647,Z 333.982,A -85,B 0,C 180,E1 -4186.755,E2 -4186.755} C_VEL
LIN {X 0,Y 530.563,Z 338.79,A -85,B 0,C 180,E1 -4187.884,E2 -4187.884} C_VEL
LIN {X 0,Y 530.51,Z 342.577,A -85,B 0,C 180,E1 -4189.035,E2 -4189.035} C_VEL
LIN {X 0,Y 530.413,Z 345.942,A -85,B 0,C 180,E1 -4190.506,E2 -4190.506} C_VEL
LIN {X 0,Y 530.383,Z 347.294,A -85,B 0,C 180,E1 -4191.48,E2 -4191.48} C_VEL
LIN {X 0,Y 530.37,Z 348.073,A -85,B 0,C 180,E1 -4192.661,E2 -4192.661} C_VEL
LIN {X 0,Y 530.407,Z 347.85,A -85,B 0,C 180,E1 -4193.926,E2 -4193.926} C_VEL
LIN {X 0,Y 530.42,Z 346.424,A -85,B 0,C 180,E1 -4195.268,E2 -4195.268} C_VEL
LIN {X 0,Y 530.489,Z 343.818,A -85,B 0,C 180,E1 -4196.578,E2 -4196.578} C_VEL
LIN {X 0,Y 530.564,Z 339.491,A -85,B 0,C 180,E1 -4198.005,E2 -4198.005} C_VEL
LIN {X 0,Y 530.671,Z 333.571,A -85,B 0,C 180,E1 -4199.41,E2 -4199.41} C_VEL
LIN {X 0,Y 530.787,Z 326.66,A -85,B 0,C 180,E1 -4200.666,E2 -4200.666} C_VEL
LIN {X 0,Y 530.975,Z 319.108,A -85,B 0,C 180,E1 -4201.759,E2 -4201.759} C_VEL
LIN {X 0,Y 531.199,Z 309.887,A -85,B 0,C 180,E1 -4202.842,E2 -4202.842} C_VEL
LIN {X 0,Y 531.474,Z 299.611,A -85,B 0,C 180,E1 -4203.811,E2 -4203.811} C_VEL
LIN {X 0,Y 531.694,Z 288.272,A -85,B 0,C 180,E1 -4204.664,E2 -4204.664} C_VEL
LIN {X 0,Y 531.96,Z 277.75,A -85,B 0,C 180,E1 -4205.291,E2 -4205.291} C_VEL
LIN {X 0,Y 532.127,Z 266.157,A -85,B 0,C 180,E1 -4205.831,E2 -4205.831} C_VEL
LIN {X 0,Y 532.341,Z 253.373,A -85,B 0,C 180,E1 -4206.255,E2 -4206.255} C_VEL
LIN {X 0,Y 532.459,Z 240.268,A -85,B 0,C 180,E1 -4206.532,E2 -4206.532} C_VEL
LIN {X 0,Y 532.731,Z 146.093,A -85,B 0,C 180,E1 -4207.822,E2 -4207.822} C_VEL
LIN {X 0,Y 531.19,Z 138.362,A -85,B 0,C 180,E1 -4207.983,E2 -4207.983} C_VEL
LIN {X 0,Y 531.301,Z 124.725,A -85,B 0,C 180,E1 -4210.689,E2 -4210.689} C_VEL
LIN {X 0,Y 531.028,Z 122.34,A -85,B 0,C 180,E1 -4211.18,E2 -4211.18} C_VEL
LIN {X 0,Y 530.987,Z 122.347,A -85,B 0,C 180,E1 -4213.862,E2 -4213.862} C_VEL
LIN {X 0,Y 530.982,Z 122.342,A -85,B 0,C 180,E1 -4216.217,E2 -4216.217} C_VEL
LIN {X 0,Y 531.036,Z 122.332,A -85,B 0,C 180,E1 -4218.55,E2 -4218.55} C_VEL
LIN {X 0,Y 531.052,Z 122.338,A -85,B 0,C 180,E1 -4221.63,E2 -4221.63} C_VEL
LIN {X 0,Y 531.121,Z 122.321,A -85,B 0,C 180,E1 -4224.685,E2 -4224.685} C_VEL
LIN {X 0,Y 531.142,Z 122.323,A -85,B 0,C 180,E1 -4227.725,E2 -4227.725} C_VEL
LIN {X 0,Y 531.15,Z 122.319,A -85,B 0,C 180,E1 -4230.758,E2 -4230.758} C_VEL
LIN {X 0,Y 531.102,Z 122.329,A -85,B 0,C 180,E1 -4233.034,E2 -4233.034} C_VEL
LIN {X 0,Y 531.075,Z 122.327,A -85,B 0,C 180,E1 -4236.077,E2 -4236.077} C_VEL
LIN {X 0,Y 531.017,Z 122.343,A -85,B 0,C 180,E1 -4239.138,E2 -4239.138} C_VEL
LIN {X 0,Y 531.041,Z 122.331,A -85,B 0,C 180,E1 -4242.225,E2 -4242.225} C_VEL
LIN {X 0,Y 530.995,Z 122.34,A -85,B 0,C 180,E1 -4245.35,E2 -4245.35} C_VEL
LIN {X 0,Y 530.984,Z 122.342,A -85,B 0,C 180,E1 -4248.521,E2 -4248.521} C_VEL
LIN {X 0,Y 530.999,Z 122.344,A -85,B 0,C 180,E1 -4250.938,E2 -4250.938} C_VEL
LIN {X 0,Y 530.971,Z 122.342,A -85,B 0,C 180,E1 -4254.225,E2 -4254.225} C_VEL
LIN {X 0,Y 531.001,Z 122.344,A -85,B 0,C 180,E1 -4256.744,E2 -4256.744} C_VEL
LIN {X 0,Y 530.98,Z 122.339,A -85,B 0,C 180,E1 -4259.323,E2 -4259.323} C_VEL
LIN {X 0,Y 530.964,Z 122.344,A -85,B 0,C 180,E1 -4262.1,E2 -4262.1} C_VEL
LIN {X 0,Y 530.967,Z 122.344,A -85,B 0,C 180,E1 -4264.851,E2 -4264.851} C_VEL
LIN {X 0,Y 530.965,Z 122.341,A -85,B 0,C 180,E1 -4267.507,E2 -4267.507} C_VEL
LIN {X 0,Y 530.98,Z 122.347,A -85,B 0,C 180,E1 -4270.433,E2 -4270.433} C_VEL
LIN {X 0,Y 530.963,Z 122.341,A -85,B 0,C 180,E1 -4273.494,E2 -4273.494} C_VEL
LIN {X 0,Y 530.957,Z 122.346,A -85,B 0,C 180,E1 -4276.505,E2 -4276.505} C_VEL
LIN {X 0,Y 530.985,Z 122.338,A -85,B 0,C 180,E1 -4278.976,E2 -4278.976} C_VEL
LIN {X 0,Y 530.957,Z 122.344,A -85,B 0,C 180,E1 -4281.529,E2 -4281.529} C_VEL
LIN {X 0,Y 530.973,Z 122.343,A -85,B 0,C 180,E1 -4284.382,E2 -4284.382} C_VEL
LIN {X 0,Y 530.965,Z 122.341,A -85,B 0,C 180,E1 -4287.133,E2 -4287.133} C_VEL
LIN {X 0,Y 530.985,Z 122.347,A -85,B 0,C 180,E1 -4289.804,E2 -4289.804} C_VEL
LIN {X 0,Y 531.01,Z 122.336,A -85,B 0,C 180,E1 -4292.468,E2 -4292.468} C_VEL
LIN {X 0,Y 530.993,Z 122.337,A -85,B 0,C 180,E1 -4294.942,E2 -4294.942} C_VEL
LIN {X 0,Y 530.969,Z 122.341,A -85,B 0,C 180,E1 -4298.247,E2 -4298.247} C_VEL
LIN {X 0,Y 530.993,Z 122.337,A -85,B 0,C 180,E1 -4300.677,E2 -4300.677} C_VEL
LIN {X 0,Y 530.984,Z 122.341,A -85,B 0,C 180,E1 -4303.071,E2 -4303.071} C_VEL
LIN {X 0,Y 531.039,Z 122.34,A -85,B 0,C 180,E1 -4305.437,E2 -4305.437} C_VEL
LIN {X 0,Y 531.035,Z 122.332,A -85,B 0,C 180,E1 -4308.55,E2 -4308.55} C_VEL
LIN {X 0,Y 531.055,Z 122.334,A -85,B 0,C 180,E1 -4311.63,E2 -4311.63} C_VEL
LIN {X 0,Y 531.123,Z 122.323,A -85,B 0,C 180,E1 -4314.685,E2 -4314.685} C_VEL
LIN {X 0,Y 531.14,Z 122.32,A -85,B 0,C 180,E1 -4317.725,E2 -4317.725} C_VEL
LIN {X 0,Y 531.151,Z 122.322,A -85,B 0,C 180,E1 -4320.758,E2 -4320.758} C_VEL
LIN {X 0,Y 531.103,Z 122.333,A -85,B 0,C 180,E1 -4323.034,E2 -4323.034} C_VEL
LIN {X 0,Y 531.075,Z 122.327,A -85,B 0,C 180,E1 -4326.077,E2 -4326.077} C_VEL
LIN {X 0,Y 531.054,Z 122.332,A -85,B 0,C 180,E1 -4328.371,E2 -4328.371} C_VEL
LIN {X 0,Y 531.05,Z 122.33,A -85,B 0,C 180,E1 -4331.672,E2 -4331.672} C_VEL
LIN {X 0,Y 531.03,Z 122.338,A -85,B 0,C 180,E1 -4334.956,E2 -4334.956} C_VEL
LIN {X 0,Y 531.016,Z 122.334,A -85,B 0,C 180,E1 -4337.723,E2 -4337.723} C_VEL
LIN {X 0,Y 530.999,Z 122.34,A -85,B 0,C 180,E1 -4340.938,E2 -4340.938} C_VEL
LIN {X 0,Y 530.971,Z 122.345,A -85,B 0,C 180,E1 -4344.225,E2 -4344.225} C_VEL
LIN {X 0,Y 531.001,Z 122.341,A -85,B 0,C 180,E1 -4346.744,E2 -4346.744} C_VEL
LIN {X 0,Y 530.981,Z 122.338,A -85,B 0,C 180,E1 -4349.323,E2 -4349.323} C_VEL
LIN {X 0,Y 530.966,Z 122.347,A -85,B 0,C 180,E1 -4352.101,E2 -4352.101} C_VEL
LIN {X 0,Y 530.97,Z 122.341,A -85,B 0,C 180,E1 -4354.851,E2 -4354.851} C_VEL
LIN {X 0,Y 530.966,Z 122.341,A -85,B 0,C 180,E1 -4357.508,E2 -4357.508} C_VEL
LIN {X 0,Y 531.027,Z 122.337,A -85,B 0,C 180,E1 -4360.429,E2 -4360.429} C_VEL
LIN {X 0,Y 530.965,Z 122.343,A -85,B 0,C 180,E1 -4363.495,E2 -4363.495} C_VEL
LIN {X 0,Y 530.966,Z 122.342,A -85,B 0,C 180,E1 -4366.506,E2 -4366.506} C_VEL
LIN {X 0,Y 531.028,Z 122.337,A -85,B 0,C 180,E1 -4369.572,E2 -4369.572} C_VEL
LIN {X 0,Y 530.969,Z 122.34,A -85,B 0,C 180,E1 -4372.577,E2 -4372.577} C_VEL
LIN {X 0,Y 530.984,Z 122.341,A -85,B 0,C 180,E1 -4375.31,E2 -4375.31} C_VEL
LIN {X 0,Y 530.969,Z 122.344,A -85,B 0,C 180,E1 -4378.032,E2 -4378.032} C_VEL
LIN {X 0,Y 530.991,Z 122.34,A -85,B 0,C 180,E1 -4380.874,E2 -4380.874} C_VEL
LIN {X 0,Y 531.004,Z 122.344,A -85,B 0,C 180,E1 -4383.256,E2 -4383.256} C_VEL
LIN {X 0,Y 531.078,Z 122.475,A -85,B 0,C 180,E1 -4384.815,E2 -4384.815} C_VEL
LIN {X 0,Y 532.471,Z 130.378,A -85,B 0,C 180,E1 -4386.055,E2 -4386.055} C_VEL
LIN {X 0,Y 532.088,Z 147.041,A -85,B 0,C 180,E1 -4388.498,E2 -4388.498} C_VEL
LIN {X 0,Y 531.786,Z 166.526,A -85,B 0,C 180,E1 -4391.308,E2 -4391.308} C_VEL
LIN {X 0,Y 531.322,Z 188.666,A -85,B 0,C 180,E1 -4394.463,E2 -4394.463} C_VEL
LIN {X 0,Y 531.281,Z 192.916,A -85,B 0,C 180,E1 -4395.046,E2 -4395.046} C_VEL
LIN {X 0,Y 532.736,Z 204.125,A -85,B 0,C 180,E1 -4395.243,E2 -4395.243} C_VEL
LIN {X 0,Y 532.375,Z 302.029,A -85,B 0,C 180,E1 -4396.594,E2 -4396.594} C_VEL
LIN {X 0,Y 532.165,Z 315.135,A -85,B 0,C 180,E1 -4396.929,E2 -4396.929} C_VEL
LIN {X 0,Y 531.929,Z 327.795,A -85,B 0,C 180,E1 -4397.408,E2 -4397.408} C_VEL
LIN {X 0,Y 531.69,Z 339.351,A -85,B 0,C 180,E1 -4398.001,E2 -4398.001} C_VEL
LIN {X 0,Y 531.441,Z 350.74,A -85,B 0,C 180,E1 -4398.752,E2 -4398.752} C_VEL
LIN {X 0,Y 531.181,Z 361.252,A -85,B 0,C 180,E1 -4399.614,E2 -4399.614} C_VEL
LIN {X 0,Y 530.974,Z 369.85,A -85,B 0,C 180,E1 -4400.477,E2 -4400.477} C_VEL
LIN {X 0,Y 530.801,Z 377.785,A -85,B 0,C 180,E1 -4401.434,E2 -4401.434} C_VEL
LIN {X 0,Y 530.665,Z 385.538,A -85,B 0,C 180,E1 -4402.581,E2 -4402.581} C_VEL
LIN {X 0,Y 530.56,Z 392.68,A -85,B 0,C 180,E1 -4403.917,E2 -4403.917} C_VEL
LIN {X 0,Y 530.459,Z 397.431,A -85,B 0,C 180,E1 -4405.06,E2 -4405.06} C_VEL
LIN {X 0,Y 530.516,Z 401.067,A -85,B 0,C 180,E1 -4406.202,E2 -4406.202} C_VEL
LIN {X 0,Y 530.512,Z 402.94,A -85,B 0,C 180,E1 -4406.962,E2 -4406.962} C_VEL
LIN {X 0,Y 530.365,Z 405.339,A -85,B 0,C 180,E1 -4408.481,E2 -4408.481} C_VEL
LIN {X 0,Y 530.362,Z 405.949,A -85,B 0,C 180,E1 -4409.241,E2 -4409.241} C_VEL
LIN {X 0,Y 530.364,Z 406.164,A -85,B 0,C 180,E1 -4410,E2 -4410} C_VEL
LIN {X 0,Y 530.362,Z 405.945,A -85,B 0,C 180,E1 -4410.759,E2 -4410.759} C_VEL
LIN {X 0,Y 530.412,Z 404.33,A -85,B 0,C 180,E1 -4412.278,E2 -4412.278} C_VEL
LIN {X 0,Y 530.512,Z 402.926,A -85,B 0,C 180,E1 -4413.037,E2 -4413.037} C_VEL
LIN {X 0,Y 530.521,Z 399.965,A -85,B 0,C 180,E1 -4414.178,E2 -4414.178} C_VEL
LIN {X 0,Y 530.522,Z 395.957,A -85,B 0,C 180,E1 -4415.321,E2 -4415.321} C_VEL
LIN {X 0,Y 530.543,Z 390.468,A -85,B 0,C 180,E1 -4416.529,E2 -4416.529} C_VEL
LIN {X 0,Y 530.681,Z 384.309,A -85,B 0,C 180,E1 -4417.61,E2 -4417.61} C_VEL
LIN {X 0,Y 530.829,Z 376.217,A -85,B 0,C 180,E1 -4418.758,E2 -4418.758} C_VEL
LIN {X 0,Y 530.995,Z 367.97,A -85,B 0,C 180,E1 -4419.715,E2 -4419.715} C_VEL
LIN {X 0,Y 531.278,Z 357.917,A -85,B 0,C 180,E1 -4420.673,E2 -4420.673} C_VEL
LIN {X 0,Y 531.507,Z 346.461,A -85,B 0,C 180,E1 -4421.543,E2 -4421.543} C_VEL
LIN {X 0,Y 531.741,Z 335.426,A -85,B 0,C 180,E1 -4422.208,E2 -4422.208} C_VEL
LIN {X 0,Y 532.001,Z 323.086,A -85,B 0,C 180,E1 -4422.784,E2 -4422.784} C_VEL
LIN {X 0,Y 532.209,Z 310.037,A -85,B 0,C 180,E1 -4423.216,E2 -4423.216} C_VEL
LIN {X 0,Y 532.415,Z 296.118,A -85,B 0,C 180,E1 -4423.502,E2 -4423.502} C_VEL
LIN {X 0,Y 532.641,Z 202.316,A -85,B 0,C 180,E1 -4424.782,E2 -4424.782} C_VEL
LIN {X 0,Y 531.247,Z 192.389,A -85,B 0,C 180,E1 -4424.968,E2 -4424.968} C_VEL
LIN {X 0,Y 531.634,Z 170.131,A -85,B 0,C 180,E1 -4428.107,E2 -4428.107} C_VEL
LIN {X 0,Y 532.039,Z 147.758,A -85,B 0,C 180,E1 -4431.301,E2 -4431.301} C_VEL
LIN {X 0,Y 532.279,Z 129.44,A -85,B 0,C 180,E1 -4433.954,E2 -4433.954} C_VEL
LIN {X 0,Y 531.069,Z 122.336,A -85,B 0,C 180,E1 -4435.054,E2 -4435.054} C_VEL
LIN {X 0,Y 531.015,Z 122.337,A -85,B 0,C 180,E1 -4437.595,E2 -4437.595} C_VEL
LIN {X 0,Y 530.976,Z 122.346,A -85,B 0,C 180,E1 -4440.645,E2 -4440.645} C_VEL
LIN {X 0,Y 530.988,Z 122.341,A -85,B 0,C 180,E1 -4443.772,E2 -4443.772} C_VEL
LIN {X 0,Y 530.956,Z 122.349,A -85,B 0,C 180,E1 -4446.558,E2 -4446.558} C_VEL
LIN {X 0,Y 531.007,Z 122.342,A -85,B 0,C 180,E1 -4449.857,E2 -4449.857} C_VEL
LIN {X 0,Y 530.981,Z 122.345,A -85,B 0,C 180,E1 -4452.456,E2 -4452.456} C_VEL
LIN {X 0,Y 530.988,Z 122.342,A -85,B 0,C 180,E1 -4455.62,E2 -4455.62} C_VEL
LIN {X 0,Y 531.008,Z 122.338,A -85,B 0,C 180,E1 -4458.565,E2 -4458.565} C_VEL
LIN {X 0,Y 530.968,Z 122.341,A -85,B 0,C 180,E1 -4461.346,E2 -4461.346} C_VEL
LIN {X 0,Y 530.953,Z 122.344,A -85,B 0,C 180,E1 -4464.38,E2 -4464.38} C_VEL
LIN {X 0,Y 530.966,Z 122.341,A -85,B 0,C 180,E1 -4467.133,E2 -4467.133} C_VEL
LIN {X 0,Y 530.969,Z 122.347,A -85,B 0,C 180,E1 -4469.803,E2 -4469.803} C_VEL
LIN {X 0,Y 531.011,Z 122.335,A -85,B 0,C 180,E1 -4472.467,E2 -4472.467} C_VEL
LIN {X 0,Y 530.994,Z 122.337,A -85,B 0,C 180,E1 -4474.942,E2 -4474.942} C_VEL
LIN {X 0,Y 530.97,Z 122.34,A -85,B 0,C 180,E1 -4478.246,E2 -4478.246} C_VEL
LIN {X 0,Y 530.994,Z 122.336,A -85,B 0,C 180,E1 -4480.677,E2 -4480.677} C_VEL
LIN {X 0,Y 530.985,Z 122.342,A -85,B 0,C 180,E1 -4483.071,E2 -4483.071} C_VEL
LIN {X 0,Y 531.039,Z 122.339,A -85,B 0,C 180,E1 -4485.436,E2 -4485.436} C_VEL
LIN {X 0,Y 531.035,Z 122.331,A -85,B 0,C 180,E1 -4488.55,E2 -4488.55} C_VEL
LIN {X 0,Y 531.055,Z 122.332,A -85,B 0,C 180,E1 -4491.629,E2 -4491.629} C_VEL
LIN {X 0,Y 531.123,Z 122.324,A -85,B 0,C 180,E1 -4494.685,E2 -4494.685} C_VEL
LIN {X 0,Y 531.14,Z 122.321,A -85,B 0,C 180,E1 -4497.725,E2 -4497.725} C_VEL
LIN {X 0,Y 531.15,Z 122.322,A -85,B 0,C 180,E1 -4500.758,E2 -4500.758} C_VEL
LIN {X 0,Y 531.103,Z 122.331,A -85,B 0,C 180,E1 -4503.034,E2 -4503.034} C_VEL
LIN {X 0,Y 531.074,Z 122.326,A -85,B 0,C 180,E1 -4506.077,E2 -4506.077} C_VEL
LIN {X 0,Y 531.053,Z 122.333,A -85,B 0,C 180,E1 -4508.37,E2 -4508.37} C_VEL
LIN {X 0,Y 531.049,Z 122.33,A -85,B 0,C 180,E1 -4511.672,E2 -4511.672} C_VEL
LIN {X 0,Y 531.028,Z 122.339,A -85,B 0,C 180,E1 -4514.956,E2 -4514.956} C_VEL
LIN {X 0,Y 531.014,Z 122.335,A -85,B 0,C 180,E1 -4517.722,E2 -4517.722} C_VEL
LIN {X 0,Y 530.998,Z 122.341,A -85,B 0,C 180,E1 -4520.938,E2 -4520.938} C_VEL
LIN {X 0,Y 530.97,Z 122.348,A -85,B 0,C 180,E1 -4524.225,E2 -4524.225} C_VEL
LIN {X 0,Y 531.004,Z 122.343,A -85,B 0,C 180,E1 -4526.744,E2 -4526.744} C_VEL
LIN {X 0,Y 530.98,Z 122.34,A -85,B 0,C 180,E1 -4529.323,E2 -4529.323} C_VEL
LIN {X 0,Y 530.978,Z 122.347,A -85,B 0,C 180,E1 -4532.103,E2 -4532.103} C_VEL
LIN {X 0,Y 531.088,Z 122.456,A -85,B 0,C 180,E1 -4534.993,E2 -4534.993} C_VEL
LIN {X 0,Y 531.358,Z 128.752,A -85,B 0,C 180,E1 -4536.215,E2 -4536.215} C_VEL
LIN {X 0,Y 531.26,Z 138.563,A -85,B 0,C 180,E1 -4538.113,E2 -4538.113} C_VEL
LIN {X 0,Y 532.821,Z 147.107,A -85,B 0,C 180,E1 -4538.281,E2 -4538.281} C_VEL
LIN {X 0,Y 532.783,Z 164.756,A -85,B 0,C 180,E1 -4538.523,E2 -4538.523} C_VEL
LIN {X 0,Y 532.154,Z 170.604,A -85,B 0,C 180,E1 -4538.585,E2 -4538.585} C_VEL
LIN {X 0,Y 526.404,Z 189.594,A -85,B 0,C 180,E1 -4538.686,E2 -4538.686} C_VEL
LIN {X 0,Y 525.786,Z 195.44,A -85,B 0,C 180,E1 -4538.751,E2 -4538.751} C_VEL
LIN {X 0,Y 525.539,Z 246.022,A -85,B 0,C 180,E1 -4539.474,E2 -4539.474} C_VEL
LIN {X 0,Y 525.33,Z 259.606,A -85,B 0,C 180,E1 -4539.834,E2 -4539.834} C_VEL
LIN {X 0,Y 525.151,Z 272.207,A -85,B 0,C 180,E1 -4540.333,E2 -4540.333} C_VEL
LIN {X 0,Y 524.896,Z 284.546,A -85,B 0,C 180,E1 -4541.001,E2 -4541.001} C_VEL
LIN {X 0,Y 524.641,Z 295.856,A -85,B 0,C 180,E1 -4541.788,E2 -4541.788} C_VEL
LIN {X 0,Y 524.404,Z 305.364,A -85,B 0,C 180,E1 -4542.612,E2 -4542.612} C_VEL
LIN {X 0,Y 524.133,Z 314.724,A -85,B 0,C 180,E1 -4543.609,E2 -4543.609} C_VEL
LIN {X 0,Y 523.86,Z 322.937,A -85,B 0,C 180,E1 -4544.681,E2 -4544.681} C_VEL
LIN {X 0,Y 523.695,Z 330.689,A -85,B 0,C 180,E1 -4545.939,E2 -4545.939} C_VEL
LIN {X 0,Y 523.562,Z 336.855,A -85,B 0,C 180,E1 -4547.228,E2 -4547.228} C_VEL
LIN {X 0,Y 523.499,Z 340.983,A -85,B 0,C 180,E1 -4548.329,E2 -4548.329} C_VEL
LIN {X 0,Y 523.415,Z 344.012,A -85,B 0,C 180,E1 -4549.367,E2 -4549.367} C_VEL
LIN {X 0,Y 523.322,Z 346.937,A -85,B 0,C 180,E1 -4550.862,E2 -4550.862} C_VEL
LIN {X 0,Y 523.291,Z 348.401,A -85,B 0,C 180,E1 -4552.409,E2 -4552.409} C_VEL
LIN {X 0,Y 523.311,Z 348.336,A -85,B 0,C 180,E1 -4553.778,E2 -4553.778} C_VEL
LIN {X 0,Y 523.297,Z 347.228,A -85,B 0,C 180,E1 -4555.009,E2 -4555.009} C_VEL
LIN {X 0,Y 523.42,Z 344.822,A -85,B 0,C 180,E1 -4556.354,E2 -4556.354} C_VEL
LIN {X 0,Y 523.481,Z 340.942,A -85,B 0,C 180,E1 -4557.758,E2 -4557.758} C_VEL
LIN {X 0,Y 523.54,Z 336.833,A -85,B 0,C 180,E1 -4558.853,E2 -4558.853} C_VEL
LIN {X 0,Y 523.687,Z 331.357,A -85,B 0,C 180,E1 -4560.007,E2 -4560.007} C_VEL
LIN {X 0,Y 523.823,Z 324.81,A -85,B 0,C 180,E1 -4561.119,E2 -4561.119} C_VEL
LIN {X 0,Y 524.042,Z 316.402,A -85,B 0,C 180,E1 -4562.268,E2 -4562.268} C_VEL
LIN {X 0,Y 524.324,Z 306.856,A -85,B 0,C 180,E1 -4563.319,E2 -4563.319} C_VEL
LIN {X 0,Y 524.581,Z 297.143,A -85,B 0,C 180,E1 -4564.189,E2 -4564.189} C_VEL
LIN {X 0,Y 524.822,Z 286.736,A -85,B 0,C 180,E1 -4564.945,E2 -4564.945} C_VEL
LIN {X 0,Y 525.081,Z 274.656,A -85,B 0,C 180,E1 -4565.63,E2 -4565.63} C_VEL
LIN {X 0,Y 525.279,Z 263.171,A -85,B 0,C 180,E1 -4566.126,E2 -4566.126} C_VEL
LIN {X 0,Y 525.482,Z 249.998,A -85,B 0,C 180,E1 -4566.528,E2 -4566.528} C_VEL
LIN {X 0,Y 525.592,Z 234.758,A -85,B 0,C 180,E1 -4566.794,E2 -4566.794} C_VEL
LIN {X 0,Y 525.944,Z 147.349,A -85,B 0,C 180,E1 -4568.004,E2 -4568.004} C_VEL
LIN {X 0,Y 524.209,Z 138.679,A -85,B 0,C 180,E1 -4568.185,E2 -4568.185} C_VEL
LIN {X 0,Y 524.341,Z 127.422,A -85,B 0,C 180,E1 -4570.422,E2 -4570.422} C_VEL
LIN {X 0,Y 523.99,Z 123.217,A -85,B 0,C 180,E1 -4571.324,E2 -4571.324} C_VEL
LIN {X 0,Y 523.938,Z 123.218,A -85,B 0,C 180,E1 -4574.438,E2 -4574.438} C_VEL
LIN {X 0,Y 523.969,Z 123.221,A -85,B 0,C 180,E1 -4577.608,E2 -4577.608} C_VEL
LIN {X 0,Y 523.939,Z 123.22,A -85,B 0,C 180,E1 -4579.958,E2 -4579.958} C_VEL
LIN {X 0,Y 524.043,Z 123.204,A -85,B 0,C 180,E1 -4582.941,E2 -4582.941} C_VEL
LIN {X 0,Y 523.967,Z 123.22,A -85,B 0,C 180,E1 -4585.384,E2 -4585.384} C_VEL
LIN {X 0,Y 524.114,Z 123.199,A -85,B 0,C 180,E1 -4587.695,E2 -4587.695} C_VEL
LIN {X 0,Y 524.121,Z 123.195,A -85,B 0,C 180,E1 -4590.768,E2 -4590.768} C_VEL
LIN {X 0,Y 524.069,Z 123.206,A -85,B 0,C 180,E1 -4593.075,E2 -4593.075} C_VEL
LIN {X 0,Y 524.034,Z 123.204,A -85,B 0,C 180,E1 -4596.159,E2 -4596.159} C_VEL
LIN {X 0,Y 523.987,Z 123.217,A -85,B 0,C 180,E1 -4599.262,E2 -4599.262} C_VEL
LIN {X 0,Y 524.003,Z 123.209,A -85,B 0,C 180,E1 -4601.739,E2 -4601.739} C_VEL
LIN {X 0,Y 523.994,Z 123.217,A -85,B 0,C 180,E1 -4605.052,E2 -4605.052} C_VEL
LIN {X 0,Y 523.947,Z 123.215,A -85,B 0,C 180,E1 -4607.969,E2 -4607.969} C_VEL
LIN {X 0,Y 523.972,Z 123.215,A -85,B 0,C 180,E1 -4610.41,E2 -4610.41} C_VEL
LIN {X 0,Y 523.911,Z 123.227,A -85,B 0,C 180,E1 -4612.893,E2 -4612.893} C_VEL
LIN {X 0,Y 523.952,Z 123.215,A -85,B 0,C 180,E1 -4615.419,E2 -4615.419} C_VEL
LIN {X 0,Y 523.964,Z 123.214,A -85,B 0,C 180,E1 -4617.999,E2 -4617.999} C_VEL
LIN {X 0,Y 523.944,Z 123.22,A -85,B 0,C 180,E1 -4620.855,E2 -4620.855} C_VEL
LIN {X 0,Y 523.929,Z 123.218,A -85,B 0,C 180,E1 -4623.729,E2 -4623.729} C_VEL
LIN {X 0,Y 523.905,Z 123.229,A -85,B 0,C 180,E1 -4626.402,E2 -4626.402} C_VEL
LIN {X 0,Y 523.919,Z 123.219,A -85,B 0,C 180,E1 -4629.085,E2 -4629.085} C_VEL
LIN {X 0,Y 523.953,Z 123.22,A -85,B 0,C 180,E1 -4632.119,E2 -4632.119} C_VEL
LIN {X 0,Y 523.953,Z 123.214,A -85,B 0,C 180,E1 -4635.309,E2 -4635.309} C_VEL
LIN {X 0,Y 523.957,Z 123.215,A -85,B 0,C 180,E1 -4638.689,E2 -4638.689} C_VEL
LIN {X 0,Y 523.918,Z 123.218,A -85,B 0,C 180,E1 -4641.08,E2 -4641.08} C_VEL
LIN {X 0,Y 523.921,Z 123.224,A -85,B 0,C 180,E1 -4643.827,E2 -4643.827} C_VEL
LIN {X 0,Y 523.94,Z 123.217,A -85,B 0,C 180,E1 -4646.636,E2 -4646.636} C_VEL
LIN {X 0,Y 523.961,Z 123.215,A -85,B 0,C 180,E1 -4649.356,E2 -4649.356} C_VEL
LIN {X 0,Y 523.975,Z 123.214,A -85,B 0,C 180,E1 -4652.281,E2 -4652.281} C_VEL
LIN {X 0,Y 523.945,Z 123.215,A -85,B 0,C 180,E1 -4654.581,E2 -4654.581} C_VEL
LIN {X 0,Y 523.917,Z 123.226,A -85,B 0,C 180,E1 -4657.756,E2 -4657.756} C_VEL
LIN {X 0,Y 523.973,Z 123.212,A -85,B 0,C 180,E1 -4660.408,E2 -4660.408} C_VEL
LIN {X 0,Y 523.965,Z 123.213,A -85,B 0,C 180,E1 -4662.837,E2 -4662.837} C_VEL
LIN {X 0,Y 524.003,Z 123.213,A -85,B 0,C 180,E1 -4665.237,E2 -4665.237} C_VEL
LIN {X 0,Y 524.011,Z 123.207,A -85,B 0,C 180,E1 -4668.394,E2 -4668.394} C_VEL
LIN {X 0,Y 524.003,Z 123.214,A -85,B 0,C 180,E1 -4671.516,E2 -4671.516} C_VEL
LIN {X 0,Y 524.084,Z 123.199,A -85,B 0,C 180,E1 -4674.614,E2 -4674.614} C_VEL
LIN {X 0,Y 524.112,Z 123.196,A -85,B 0,C 180,E1 -4677.695,E2 -4677.695} C_VEL
LIN {X 0,Y 524.121,Z 123.198,A -85,B 0,C 180,E1 -4680.768,E2 -4680.768} C_VEL
LIN {X 0,Y 524.07,Z 123.208,A -85,B 0,C 180,E1 -4683.075,E2 -4683.075} C_VEL
LIN {X 0,Y 524.037,Z 123.204,A -85,B 0,C 180,E1 -4686.159,E2 -4686.159} C_VEL
LIN {X 0,Y 524.002,Z 123.211,A -85,B 0,C 180,E1 -4688.484,E2 -4688.484} C_VEL
LIN {X 0,Y 524.002,Z 123.208,A -85,B 0,C 180,E1 -4691.74,E2 -4691.74} C_VEL
LIN {X 0,Y 523.992,Z 123.213,A -85,B 0,C 180,E1 -4695.053,E2 -4695.053} C_VEL
LIN {X 0,Y 523.963,Z 123.214,A -85,B 0,C 180,E1 -4697.969,E2 -4697.969} C_VEL
LIN {X 0,Y 523.971,Z 123.218,A -85,B 0,C 180,E1 -4700.41,E2 -4700.41} C_VEL
LIN {X 0,Y 523.91,Z 123.223,A -85,B 0,C 180,E1 -4702.894,E2 -4702.894} C_VEL
LIN {X 0,Y 523.952,Z 123.214,A -85,B 0,C 180,E1 -4705.419,E2 -4705.419} C_VEL
LIN {X 0,Y 523.967,Z 123.216,A -85,B 0,C 180,E1 -4707.999,E2 -4707.999} C_VEL
LIN {X 0,Y 523.944,Z 123.217,A -85,B 0,C 180,E1 -4710.855,E2 -4710.855} C_VEL
LIN {X 0,Y 523.959,Z 123.215,A -85,B 0,C 180,E1 -4713.735,E2 -4713.735} C_VEL
LIN {X 0,Y 523.903,Z 123.226,A -85,B 0,C 180,E1 -4716.402,E2 -4716.402} C_VEL
LIN {X 0,Y 523.932,Z 123.217,A -85,B 0,C 180,E1 -4719.084,E2 -4719.084} C_VEL
LIN {X 0,Y 523.973,Z 123.212,A -85,B 0,C 180,E1 -4721.313,E2 -4721.313} C_VEL
LIN {X 0,Y 523.957,Z 123.214,A -85,B 0,C 180,E1 -4724.692,E2 -4724.692} C_VEL
LIN {X 0,Y 523.958,Z 123.222,A -85,B 0,C 180,E1 -4727.882,E2 -4727.882} C_VEL
LIN {X 0,Y 523.98,Z 123.219,A -85,B 0,C 180,E1 -4729.924,E2 -4729.924} C_VEL
LIN {X 0,Y 523.909,Z 123.22,A -85,B 0,C 180,E1 -4732.868,E2 -4732.868} C_VEL
LIN {X 0,Y 523.934,Z 123.226,A -85,B 0,C 180,E1 -4735.71,E2 -4735.71} C_VEL
LIN {X 0,Y 523.923,Z 123.218,A -85,B 0,C 180,E1 -4738.456,E2 -4738.456} C_VEL
LIN {X 0,Y 523.941,Z 123.221,A -85,B 0,C 180,E1 -4741.126,E2 -4741.126} C_VEL
LIN {X 0,Y 523.987,Z 123.218,A -85,B 0,C 180,E1 -4743.981,E2 -4743.981} C_VEL
LIN {X 0,Y 524.009,Z 123.336,A -85,B 0,C 180,E1 -4744.638,E2 -4744.638} C_VEL
LIN {X 0,Y 525.513,Z 131.42,A -85,B 0,C 180,E1 -4745.927,E2 -4745.927} C_VEL
LIN {X 0,Y 525.144,Z 146.711,A -85,B 0,C 180,E1 -4748.2,E2 -4748.2} C_VEL
LIN {X 0,Y 524.802,Z 163.371,A -85,B 0,C 180,E1 -4750.644,E2 -4750.644} C_VEL
LIN {X 0,Y 524.46,Z 182.767,A -85,B 0,C 180,E1 -4753.456,E2 -4753.456} C_VEL
LIN {X 0,Y 524.258,Z 192.584,A -85,B 0,C 180,E1 -4754.842,E2 -4754.842} C_VEL
LIN {X 0,Y 525.855,Z 205.216,A -85,B 0,C 180,E1 -4755.066,E2 -4755.066} C_VEL
LIN {X 0,Y 525.479,Z 301.513,A -85,B 0,C 180,E1 -4756.415,E2 -4756.415} C_VEL
LIN {X 0,Y 525.247,Z 314.661,A -85,B 0,C 180,E1 -4756.754,E2 -4756.754} C_VEL
LIN {X 0,Y 524.997,Z 327.346,A -85,B 0,C 180,E1 -4757.239,E2 -4757.239} C_VEL
LIN {X 0,Y 524.69,Z 339.436,A -85,B 0,C 180,E1 -4757.871,E2 -4757.871} C_VEL
LIN {X 0,Y 524.387,Z 351.618,A -85,B 0,C 180,E1 -4758.696,E2 -4758.696} C_VEL
LIN {X 0,Y 524.129,Z 361.899,A -85,B 0,C 180,E1 -4759.571,E2 -4759.571} C_VEL
LIN {X 0,Y 523.879,Z 371.141,A -85,B 0,C 180,E1 -4760.541,E2 -4760.541} C_VEL
LIN {X 0,Y 523.674,Z 380.144,A -85,B 0,C 180,E1 -4761.705,E2 -4761.705} C_VEL
LIN {X 0,Y 523.568,Z 387.396,A -85,B 0,C 180,E1 -4762.867,E2 -4762.867} C_VEL
LIN {X 0,Y 523.457,Z 392.287,A -85,B 0,C 180,E1 -4763.834,E2 -4763.834} C_VEL
LIN {X 0,Y 523.383,Z 397.042,A -85,B 0,C 180,E1 -4764.993,E2 -4764.993} C_VEL
LIN {X 0,Y 523.443,Z 400.68,A -85,B 0,C 180,E1 -4766.151,E2 -4766.151} C_VEL
LIN {X 0,Y 523.417,Z 402.553,A -85,B 0,C 180,E1 -4766.921,E2 -4766.921} C_VEL
LIN {X 0,Y 523.338,Z 403.954,A -85,B 0,C 180,E1 -4767.691,E2 -4767.691} C_VEL
LIN {X 0,Y 523.272,Z 405.562,A -85,B 0,C 180,E1 -4769.23,E2 -4769.23} C_VEL
LIN {X 0,Y 523.275,Z 405.777,A -85,B 0,C 180,E1 -4770,E2 -4770} C_VEL
LIN {X 0,Y 523.272,Z 405.556,A -85,B 0,C 180,E1 -4770.77,E2 -4770.77} C_VEL
LIN {X 0,Y 523.338,Z 403.938,A -85,B 0,C 180,E1 -4772.309,E2 -4772.309} C_VEL
LIN {X 0,Y 523.417,Z 402.53,A -85,B 0,C 180,E1 -4773.079,E2 -4773.079} C_VEL
LIN {X 0,Y 523.423,Z 399.565,A -85,B 0,C 180,E1 -4774.235,E2 -4774.235} C_VEL
LIN {X 0,Y 523.455,Z 395.553,A -85,B 0,C 180,E1 -4775.393,E2 -4775.393} C_VEL
LIN {X 0,Y 523.501,Z 389.466,A -85,B 0,C 180,E1 -4776.73,E2 -4776.73} C_VEL
LIN {X 0,Y 523.644,Z 382.646,A -85,B 0,C 180,E1 -4777.907,E2 -4777.907} C_VEL
LIN {X 0,Y 523.819,Z 374.286,A -85,B 0,C 180,E1 -4779.07,E2 -4779.07} C_VEL
LIN {X 0,Y 523.993,Z 365.712,A -85,B 0,C 180,E1 -4780.041,E2 -4780.041} C_VEL
LIN {X 0,Y 524.288,Z 355.13,A -85,B 0,C 180,E1 -4781.012,E2 -4781.012} C_VEL
LIN {X 0,Y 524.549,Z 343.469,A -85,B 0,C 180,E1 -4781.871,E2 -4781.871} C_VEL
LIN {X 0,Y 524.897,Z 331.206,A -85,B 0,C 180,E1 -4782.567,E2 -4782.567} C_VEL
LIN {X 0,Y 525.096,Z 318.707,A -85,B 0,C 180,E1 -4783.102,E2 -4783.102} C_VEL
LIN {X 0,Y 525.374,Z 305.782,A -85,B 0,C 180,E1 -4783.489,E2 -4783.489} C_VEL
LIN {X 0,Y 525.569,Z 290.259,A -85,B 0,C 180,E1 -4783.755,E2 -4783.755} C_VEL
LIN {X 0,Y 525.691,Z 202.53,A -85,B 0,C 180,E1 -4784.973,E2 -4784.973} C_VEL
LIN {X 0,Y 524.231,Z 191.951,A -85,B 0,C 180,E1 -4785.175,E2 -4785.175} C_VEL
LIN {X 0,Y 524.635,Z 170.039,A -85,B 0,C 180,E1 -4788.308,E2 -4788.308} C_VEL
LIN {X 0,Y 525.057,Z 148.725,A -85,B 0,C 180,E1 -4791.392,E2 -4791.392} C_VEL
LIN {X 0,Y 525.372,Z 131.844,A -85,B 0,C 180,E1 -4793.867,E2 -4793.867} C_VEL
LIN {X 0,Y 524.3,Z 124.689,A -85,B 0,C 180,E1 -4794.976,E2 -4794.976} C_VEL
LIN {X 0,Y 524.005,Z 123.215,A -85,B 0,C 180,E1 -4795.23,E2 -4795.23} C_VEL
LIN {X 0,Y 523.97,Z 123.218,A -85,B 0,C 180,E1 -4797.999,E2 -4797.999} C_VEL
LIN {X 0,Y 523.946,Z 123.219,A -85,B 0,C 180,E1 -4800.854,E2 -4800.854} C_VEL
LIN {X 0,Y 523.96,Z 123.217,A -85,B 0,C 180,E1 -4803.734,E2 -4803.734} C_VEL
LIN {X 0,Y 523.904,Z 123.229,A -85,B 0,C 180,E1 -4806.401,E2 -4806.401} C_VEL
LIN {X 0,Y 523.933,Z 123.219,A -85,B 0,C 180,E1 -4809.083,E2 -4809.083} C_VEL
LIN {X 0,Y 523.974,Z 123.213,A -85,B 0,C 180,E1 -4811.312,E2 -4811.312} C_VEL
LIN {X 0,Y 523.956,Z 123.217,A -85,B 0,C 180,E1 -4814.691,E2 -4814.691} C_VEL
LIN {X 0,Y 523.957,Z 123.223,A -85,B 0,C 180,E1 -4817.881,E2 -4817.881} C_VEL
LIN {X 0,Y 523.979,Z 123.22,A -85,B 0,C 180,E1 -4819.923,E2 -4819.923} C_VEL
LIN {X 0,Y 523.907,Z 123.221,A -85,B 0,C 180,E1 -4822.867,E2 -4822.867} C_VEL
LIN {X 0,Y 523.932,Z 123.224,A -85,B 0,C 180,E1 -4825.709,E2 -4825.709} C_VEL
LIN {X 0,Y 523.92,Z 123.22,A -85,B 0,C 180,E1 -4828.456,E2 -4828.456} C_VEL
LIN {X 0,Y 523.937,Z 123.216,A -85,B 0,C 180,E1 -4831.125,E2 -4831.125} C_VEL
LIN {X 0,Y 523.983,Z 123.214,A -85,B 0,C 180,E1 -4833.98,E2 -4833.98} C_VEL
LIN {X 0,Y 523.909,Z 123.221,A -85,B 0,C 180,E1 -4837.106,E2 -4837.106} C_VEL
LIN {X 0,Y 523.978,Z 123.214,A -85,B 0,C 180,E1 -4839.866,E2 -4839.866} C_VEL
LIN {X 0,Y 523.965,Z 123.214,A -85,B 0,C 180,E1 -4842.837,E2 -4842.837} C_VEL
LIN {X 0,Y 524.003,Z 123.213,A -85,B 0,C 180,E1 -4845.236,E2 -4845.236} C_VEL
LIN {X 0,Y 524.011,Z 123.206,A -85,B 0,C 180,E1 -4848.394,E2 -4848.394} C_VEL
LIN {X 0,Y 524.003,Z 123.212,A -85,B 0,C 180,E1 -4851.516,E2 -4851.516} C_VEL
LIN {X 0,Y 524.084,Z 123.2,A -85,B 0,C 180,E1 -4854.614,E2 -4854.614} C_VEL
LIN {X 0,Y 524.112,Z 123.196,A -85,B 0,C 180,E1 -4857.694,E2 -4857.694} C_VEL
LIN {X 0,Y 524.121,Z 123.197,A -85,B 0,C 180,E1 -4860.768,E2 -4860.768} C_VEL
LIN {X 0,Y 524.07,Z 123.207,A -85,B 0,C 180,E1 -4863.075,E2 -4863.075} C_VEL
LIN {X 0,Y 524.036,Z 123.204,A -85,B 0,C 180,E1 -4866.159,E2 -4866.159} C_VEL
